LIN {X 0,Y 115.903,Z 1227.166,A -85,B 0,C 180,E1 30525.083,E2 30525.083} C_VEL
LIN {X 0,Y 121.307,Z 1221.826,A -85,B 0,C 180,E1 30544.058,E2 30544.058} C_VEL
LIN {X 0,Y 149.236,Z 1207.445,A -85,B 0,C 180,E1 30568.46,E2 30568.46} C_VEL
LIN {X 0,Y 160.737,Z 1202.235,A -85,B 0,C 180,E1 30574.059,E2 30574.059} C_VEL
LIN {X 0,Y 129.923,Z 1200.348,A -85,B 0,C 180,E1 30593.319,E2 30593.319} C_VEL
LIN {X 0,Y 116.524,Z 1195.812,A -85,B 0,C 180,E1 30615.028,E2 30615.028} C_VEL
LIN {X 0,Y 115.852,Z 1188.978,A -85,B 0,C 180,E1 30635.424,E2 30635.424} C_VEL
LIN {X 0,Y 122.473,Z 1180.721,A -85,B 0,C 180,E1 30651.947,E2 30651.947} C_VEL
LIN {X 0,Y 138.737,Z 1166.544,A -85,B 0,C 180,E1 30669.914,E2 30669.914} C_VEL
LIN {X 0,Y 165.96,Z 1145.332,A -85,B 0,C 180,E1 30684.797,E2 30684.797} C_VEL
LIN {X 0,Y 197.116,Z 1119.047,A -85,B 0,C 180,E1 30694.805,E2 30694.805} C_VEL
LIN {X 0,Y 228.825,Z 1088.466,A -85,B 0,C 180,E1 30701.734,E2 30701.734} C_VEL
LIN {X 0,Y 247.509,Z 1067.925,A -85,B 0,C 180,E1 30704.862,E2 30704.862} C_VEL
LIN {X 0,Y 250.073,Z 1055.769,A -85,B 0,C 180,E1 30711.272,E2 30711.272} C_VEL
LIN {X 0,Y 251.256,Z 1045.915,A -85,B 0,C 180,E1 30717.768,E2 30717.768} C_VEL
LIN {X 0,Y 251.874,Z 1037.298,A -85,B 0,C 180,E1 30725.345,E2 30725.345} C_VEL
LIN {X 0,Y 252.29,Z 1032.887,A -85,B 0,C 180,E1 30731.229,E2 30731.229} C_VEL
LIN {X 0,Y 252.785,Z 1030.009,A -85,B 0,C 180,E1 30738.891,E2 30738.891} C_VEL
LIN {X 0,Y 253.685,Z 1029.517,A -85,B 0,C 180,E1 30744.152,E2 30744.152} C_VEL
LIN {X 0,Y 252.999,Z 1031.73,A -85,B 0,C 180,E1 30747.067,E2 30747.067} C_VEL
LIN {X 0,Y 251.361,Z 1037.125,A -85,B 0,C 180,E1 30751.921,E2 30751.921} C_VEL
LIN {X 0,Y 254.488,Z 1040.821,A -85,B 0,C 180,E1 30759.132,E2 30759.132} C_VEL
LIN {X 0,Y 258.114,Z 1049.252,A -85,B 0,C 180,E1 30767.246,E2 30767.246} C_VEL
LIN {X 0,Y 260.709,Z 1059.906,A -85,B 0,C 180,E1 30773.967,E2 30773.967} C_VEL
LIN {X 0,Y 263.22,Z 1075.308,A -85,B 0,C 180,E1 30781.406,E2 30781.406} C_VEL
LIN {X 0,Y 263.374,Z 1076.931,A -85,B 0,C 180,E1 30782.108,E2 30782.108} C_VEL
LIN {X 0,Y 229.491,Z 1117.049,A -85,B 0,C 180,E1 30786.492,E2 30786.492} C_VEL
LIN {X 0,Y 196.364,Z 1149.598,A -85,B 0,C 180,E1 30792.406,E2 30792.406} C_VEL
LIN {X 0,Y 164.117,Z 1177.145,A -85,B 0,C 180,E1 30801.157,E2 30801.157} C_VEL
LIN {X 0,Y 136.729,Z 1198.115,A -85,B 0,C 180,E1 30813.545,E2 30813.545} C_VEL
LIN {X 0,Y 117.332,Z 1213.51,A -85,B 0,C 180,E1 30830.599,E2 30830.599} C_VEL
LIN {X 0,Y 109.107,Z 1222.749,A -85,B 0,C 180,E1 30849.709,E2 30849.709} C_VEL
LIN {X 0,Y 108.282,Z 1226.006,A -85,B 0,C 180,E1 30861.945,E2 30861.945} C_VEL
LIN {X 0,Y 109.205,Z 1227.073,A -85,B 0,C 180,E1 30869.968,E2 30869.968} C_VEL
LIN {X 0,Y 108.146,Z 1225.726,A -85,B 0,C 180,E1 30886.193,E2 30886.193} C_VEL
LIN {X 0,Y 115.945,Z 1219.699,A -85,B 0,C 180,E1 30908.559,E2 30908.559} C_VEL
LIN {X 0,Y 148.879,Z 1205.076,A -85,B 0,C 180,E1 30933.089,E2 30933.089} C_VEL
LIN {X 0,Y 150.497,Z 1204.236,A -85,B 0,C 180,E1 30934.137,E2 30934.137} C_VEL
LIN {X 0,Y 121.73,Z 1201.678,A -85,B 0,C 180,E1 30952.998,E2 30952.998} C_VEL
LIN {X 0,Y 108.299,Z 1196.353,A -85,B 0,C 180,E1 30976.2,E2 30976.2} C_VEL
LIN {X 0,Y 108.593,Z 1188.984,A -85,B 0,C 180,E1 30997.991,E2 30997.991} C_VEL
LIN {X 0,Y 116.696,Z 1180.045,A -85,B 0,C 180,E1 31015.734,E2 31015.734} C_VEL
LIN {X 0,Y 137.512,Z 1163.474,A -85,B 0,C 180,E1 31035.364,E2 31035.364} C_VEL
LIN {X 0,Y 166.233,Z 1141.644,A -85,B 0,C 180,E1 31048.906,E2 31048.906} C_VEL
LIN {X 0,Y 198.392,Z 1114.848,A -85,B 0,C 180,E1 31058.079,E2 31058.079} C_VEL
LIN {X 0,Y 232.591,Z 1081.271,A -85,B 0,C 180,E1 31064.742,E2 31064.742} C_VEL
LIN {X 0,Y 242.121,Z 1070.542,A -85,B 0,C 180,E1 31066.39,E2 31066.39} C_VEL
LIN {X 0,Y 244.698,Z 1059.241,A -85,B 0,C 180,E1 31072.716,E2 31072.716} C_VEL
LIN {X 0,Y 245.996,Z 1049.786,A -85,B 0,C 180,E1 31079.449,E2 31079.449} C_VEL
LIN {X 0,Y 247.016,Z 1041.487,A -85,B 0,C 180,E1 31087.732,E2 31087.732} C_VEL
LIN {X 0,Y 247.351,Z 1038.331,A -85,B 0,C 180,E1 31092.86,E2 31092.86} C_VEL
LIN {X 0,Y 248.6,Z 1035.925,A -85,B 0,C 180,E1 31102.224,E2 31102.224} C_VEL
LIN {X 0,Y 251.159,Z 1036.873,A -85,B 0,C 180,E1 31111.232,E2 31111.232} C_VEL
LIN {X 0,Y 251.361,Z 1037.125,A -85,B 0,C 180,E1 31111.921,E2 31111.921} C_VEL
LIN {X 0,Y 251.021,Z 1040.302,A -85,B 0,C 180,E1 31114.822,E2 31114.822} C_VEL
LIN {X 0,Y 249.783,Z 1047.533,A -85,B 0,C 180,E1 31119.608,E2 31119.608} C_VEL
LIN {X 0,Y 253.284,Z 1056.269,A -85,B 0,C 180,E1 31127.95,E2 31127.95} C_VEL
LIN {X 0,Y 255.662,Z 1067.949,A -85,B 0,C 180,E1 31135.014,E2 31135.014} C_VEL
LIN {X 0,Y 256.974,Z 1080.351,A -85,B 0,C 180,E1 31140.941,E2 31140.941} C_VEL
LIN {X 0,Y 223.473,Z 1118.609,A -85,B 0,C 180,E1 31145.07,E2 31145.07} C_VEL
LIN {X 0,Y 186.796,Z 1153.281,A -85,B 0,C 180,E1 31151.557,E2 31151.557} C_VEL
LIN {X 0,Y 154.639,Z 1179.212,A -85,B 0,C 180,E1 31160.504,E2 31160.504} C_VEL
LIN {X 0,Y 127.088,Z 1199.404,A -85,B 0,C 180,E1 31173.616,E2 31173.616} C_VEL
LIN {X 0,Y 108.285,Z 1213.812,A -85,B 0,C 180,E1 31191.784,E2 31191.784} C_VEL
LIN {X 0,Y 100.902,Z 1222.307,A -85,B 0,C 180,E1 31212.535,E2 31212.535} C_VEL
LIN {X 0,Y 101.407,Z 1225.453,A -85,B 0,C 180,E1 31229.965,E2 31229.965} C_VEL
LIN {X 0,Y 100.398,Z 1224.298,A -85,B 0,C 180,E1 31247.481,E2 31247.481} C_VEL
LIN {X 0,Y 107.237,Z 1219.449,A -85,B 0,C 180,E1 31267.89,E2 31267.89} C_VEL
LIN {X 0,Y 136.554,Z 1207.341,A -85,B 0,C 180,E1 31292.225,E2 31292.225} C_VEL
LIN {X 0,Y 139.784,Z 1205.877,A -85,B 0,C 180,E1 31294.379,E2 31294.379} C_VEL
LIN {X 0,Y 107.624,Z 1201.286,A -85,B 0,C 180,E1 31319.997,E2 31319.997} C_VEL
LIN {X 0,Y 99.274,Z 1194.993,A -85,B 0,C 180,E1 31344.128,E2 31344.128} C_VEL
LIN {X 0,Y 103.71,Z 1186.418,A -85,B 0,C 180,E1 31366.753,E2 31366.753} C_VEL
LIN {X 0,Y 116.196,Z 1175.396,A -85,B 0,C 180,E1 31385.536,E2 31385.536} C_VEL
LIN {X 0,Y 141.482,Z 1157.033,A -85,B 0,C 180,E1 31402.985,E2 31402.985} C_VEL
LIN {X 0,Y 172.324,Z 1133.681,A -85,B 0,C 180,E1 31414.551,E2 31414.551} C_VEL
LIN {X 0,Y 205.729,Z 1105.109,A -85,B 0,C 180,E1 31422.412,E2 31422.412} C_VEL
LIN {X 0,Y 236.572,Z 1073.596,A -85,B 0,C 180,E1 31427.744,E2 31427.744} C_VEL
LIN {X 0,Y 239.332,Z 1062.684,A -85,B 0,C 180,E1 31434.245,E2 31434.245} C_VEL
LIN {X 0,Y 240.84,Z 1053.518,A -85,B 0,C 180,E1 31441.491,E2 31441.491} C_VEL
LIN {X 0,Y 241.954,Z 1046.947,A -85,B 0,C 180,E1 31448.665,E2 31448.665} C_VEL
LIN {X 0,Y 242.687,Z 1043.093,A -85,B 0,C 180,E1 31456.777,E2 31456.777} C_VEL
LIN {X 0,Y 244.616,Z 1042.241,A -85,B 0,C 180,E1 31466.227,E2 31466.227} C_VEL
LIN {X 0,Y 247.713,Z 1044.501,A -85,B 0,C 180,E1 31474.725,E2 31474.725} C_VEL
LIN {X 0,Y 249.783,Z 1047.533,A -85,B 0,C 180,E1 31479.608,E2 31479.608} C_VEL
LIN {X 0,Y 249.353,Z 1051.979,A -85,B 0,C 180,E1 31482.44,E2 31482.44} C_VEL
LIN {X 0,Y 247.711,Z 1061.226,A -85,B 0,C 180,E1 31487.083,E2 31487.083} C_VEL
LIN {X 0,Y 249.801,Z 1071.906,A -85,B 0,C 180,E1 31493.925,E2 31493.925} C_VEL
LIN {X 0,Y 251.125,Z 1082.686,A -85,B 0,C 180,E1 31499.497,E2 31499.497} C_VEL
LIN {X 0,Y 220.201,Z 1117.408,A -85,B 0,C 180,E1 31503.214,E2 31503.214} C_VEL
LIN {X 0,Y 182.355,Z 1152.44,A -85,B 0,C 180,E1 31509.541,E2 31509.541} C_VEL
LIN {X 0,Y 148.605,Z 1178.767,A -85,B 0,C 180,E1 31518.583,E2 31518.583} C_VEL
LIN {X 0,Y 120.171,Z 1198.668,A -85,B 0,C 180,E1 31531.868,E2 31531.868} C_VEL
LIN {X 0,Y 101.316,Z 1212.21,A -85,B 0,C 180,E1 31549.776,E2 31549.776} C_VEL
LIN {X 0,Y 93.27,Z 1220.523,A -85,B 0,C 180,E1 31571.054,E2 31571.054} C_VEL
LIN {X 0,Y 93.589,Z 1223.855,A -85,B 0,C 180,E1 31589.962,E2 31589.962} C_VEL
LIN {X 0,Y 92.711,Z 1222.762,A -85,B 0,C 180,E1 31608.984,E2 31608.984} C_VEL
LIN {X 0,Y 104.857,Z 1216.407,A -85,B 0,C 180,E1 31636.049,E2 31636.049} C_VEL
LIN {X 0,Y 129.649,Z 1207.413,A -85,B 0,C 180,E1 31654.348,E2 31654.348} C_VEL
LIN {X 0,Y 99.287,Z 1202.08,A -85,B 0,C 180,E1 31679.997,E2 31679.997} C_VEL
LIN {X 0,Y 91.371,Z 1195.363,A -85,B 0,C 180,E1 31705.839,E2 31705.839} C_VEL
LIN {X 0,Y 96.333,Z 1187.072,A -85,B 0,C 180,E1 31728.41,E2 31728.41} C_VEL
LIN {X 0,Y 110.812,Z 1175.137,A -85,B 0,C 180,E1 31748.955,E2 31748.955} C_VEL
LIN {X 0,Y 137.994,Z 1156.444,A -85,B 0,C 180,E1 31766.214,E2 31766.214} C_VEL
LIN {X 0,Y 171.971,Z 1131.211,A -85,B 0,C 180,E1 31777.815,E2 31777.815} C_VEL
LIN {X 0,Y 205.821,Z 1102.143,A -85,B 0,C 180,E1 31785.048,E2 31785.048} C_VEL
LIN {X 0,Y 231.083,Z 1076.83,A -85,B 0,C 180,E1 31789.1,E2 31789.1} C_VEL
LIN {X 0,Y 234.064,Z 1066.08,A -85,B 0,C 180,E1 31795.989,E2 31795.989} C_VEL
LIN {X 0,Y 235.794,Z 1057.293,A -85,B 0,C 180,E1 31803.589,E2 31803.589} C_VEL
LIN {X 0,Y 236.788,Z 1052.096,A -85,B 0,C 180,E1 31810.029,E2 31810.029} C_VEL
LIN {X 0,Y 237.495,Z 1049.645,A -85,B 0,C 180,E1 31815.588,E2 31815.588} C_VEL
LIN {X 0,Y 239.297,Z 1048.305,A -85,B 0,C 180,E1 31825.2,E2 31825.2} C_VEL
LIN {X 0,Y 242.39,Z 1050.363,A -85,B 0,C 180,E1 31834.13,E2 31834.13} C_VEL
LIN {X 0,Y 244.886,Z 1053.918,A -85,B 0,C 180,E1 31840.029,E2 31840.029} C_VEL
LIN {X 0,Y 247.711,Z 1061.226,A -85,B 0,C 180,E1 31847.083,E2 31847.083} C_VEL
LIN {X 0,Y 246.931,Z 1067.057,A -85,B 0,C 180,E1 31849.812,E2 31849.812} C_VEL
LIN {X 0,Y 244.195,Z 1078.298,A -85,B 0,C 180,E1 31854.237,E2 31854.237} C_VEL
LIN {X 0,Y 244.491,Z 1086.498,A -85,B 0,C 180,E1 31858.263,E2 31858.263} C_VEL
LIN {X 0,Y 209.883,Z 1123.195,A -85,B 0,C 180,E1 31862.262,E2 31862.262} C_VEL
LIN {X 0,Y 174.487,Z 1154.462,A -85,B 0,C 180,E1 31868.179,E2 31868.179} C_VEL
LIN {X 0,Y 139.774,Z 1180.356,A -85,B 0,C 180,E1 31877.532,E2 31877.532} C_VEL
LIN {X 0,Y 110.922,Z 1199.471,A -85,B 0,C 180,E1 31891.574,E2 31891.574} C_VEL
LIN {X 0,Y 90.556,Z 1213.571,A -85,B 0,C 180,E1 31914.224,E2 31914.224} C_VEL
LIN {X 0,Y 84.916,Z 1220.325,A -85,B 0,C 180,E1 31936.947,E2 31936.947} C_VEL
LIN {X 0,Y 85.769,Z 1222.218,A -85,B 0,C 180,E1 31949.959,E2 31949.959} C_VEL
LIN {X 0,Y 85.128,Z 1221.178,A -85,B 0,C 180,E1 31970.749,E2 31970.749} C_VEL
LIN {X 0,Y 99.219,Z 1215.064,A -85,B 0,C 180,E1 31999.539,E2 31999.539} C_VEL
LIN {X 0,Y 118.108,Z 1208.948,A -85,B 0,C 180,E1 32013.513,E2 32013.513} C_VEL
LIN {X 0,Y 118.736,Z 1208.442,A -85,B 0,C 180,E1 32014.648,E2 32014.648} C_VEL
LIN {X 0,Y 90.605,Z 1202.768,A -85,B 0,C 180,E1 32040.532,E2 32040.532} C_VEL
LIN {X 0,Y 83.576,Z 1195.469,A -85,B 0,C 180,E1 32068.735,E2 32068.735} C_VEL
LIN {X 0,Y 90.422,Z 1186.476,A -85,B 0,C 180,E1 32093.096,E2 32093.096} C_VEL
LIN {X 0,Y 109.279,Z 1172.666,A -85,B 0,C 180,E1 32115.427,E2 32115.427} C_VEL
LIN {X 0,Y 138.694,Z 1153.021,A -85,B 0,C 180,E1 32131.101,E2 32131.101} C_VEL
LIN {X 0,Y 171.661,Z 1128.922,A -85,B 0,C 180,E1 32140.994,E2 32140.994} C_VEL
LIN {X 0,Y 209.084,Z 1096.491,A -85,B 0,C 180,E1 32148.146,E2 32148.146} C_VEL
LIN {X 0,Y 225.667,Z 1079.947,A -85,B 0,C 180,E1 32150.598,E2 32150.598} C_VEL
LIN {X 0,Y 228.771,Z 1069.776,A -85,B 0,C 180,E1 32157.556,E2 32157.556} C_VEL
LIN {X 0,Y 230.922,Z 1060.913,A -85,B 0,C 180,E1 32166.099,E2 32166.099} C_VEL
LIN {X 0,Y 232.082,Z 1056.025,A -85,B 0,C 180,E1 32174.263,E2 32174.263} C_VEL
LIN {X 0,Y 233.247,Z 1054.561,A -85,B 0,C 180,E1 32181.047,E2 32181.047} C_VEL
LIN {X 0,Y 235.455,Z 1054.955,A -85,B 0,C 180,E1 32189.112,E2 32189.112} C_VEL
LIN {X 0,Y 238.834,Z 1058.342,A -85,B 0,C 180,E1 32197.693,E2 32197.693} C_VEL
LIN {X 0,Y 241.94,Z 1065.38,A -85,B 0,C 180,E1 32205.535,E2 32205.535} C_VEL
LIN {X 0,Y 243.76,Z 1074.732,A -85,B 0,C 180,E1 32212.154,E2 32212.154} C_VEL
LIN {X 0,Y 244.195,Z 1078.298,A -85,B 0,C 180,E1 32214.237,E2 32214.237} C_VEL
LIN {X 0,Y 242.463,Z 1083.265,A -85,B 0,C 180,E1 32215.784,E2 32215.784} C_VEL
LIN {X 0,Y 235.136,Z 1093.065,A -85,B 0,C 180,E1 32217.169,E2 32217.169} C_VEL
LIN {X 0,Y 225.579,Z 1103.372,A -85,B 0,C 180,E1 32218.121,E2 32218.121} C_VEL
LIN {X 0,Y 187.741,Z 1139.371,A -85,B 0,C 180,E1 32222.924,E2 32222.924} C_VEL
LIN {X 0,Y 150.886,Z 1168.156,A -85,B 0,C 180,E1 32230.295,E2 32230.295} C_VEL
LIN {X 0,Y 117.953,Z 1190.195,A -85,B 0,C 180,E1 32241.676,E2 32241.676} C_VEL
LIN {X 0,Y 89.807,Z 1207.468,A -85,B 0,C 180,E1 32262.303,E2 32262.303} C_VEL
LIN {X 0,Y 78.256,Z 1216.707,A -85,B 0,C 180,E1 32287.234,E2 32287.234} C_VEL
LIN {X 0,Y 77.955,Z 1220.615,A -85,B 0,C 180,E1 32309.955,E2 32309.955} C_VEL
LIN {X 0,Y 77.617,Z 1219.589,A -85,B 0,C 180,E1 32332.865,E2 32332.865} C_VEL
LIN {X 0,Y 93.973,Z 1213.764,A -85,B 0,C 180,E1 32363.449,E2 32363.449} C_VEL
LIN {X 0,Y 107.273,Z 1209.979,A -85,B 0,C 180,E1 32373.353,E2 32373.353} C_VEL
LIN {X 0,Y 107.65,Z 1209.322,A -85,B 0,C 180,E1 32375.094,E2 32375.094} C_VEL
LIN {X 0,Y 82.522,Z 1203.513,A -85,B 0,C 180,E1 32399.996,E2 32399.996} C_VEL
LIN {X 0,Y 75.939,Z 1195.293,A -85,B 0,C 180,E1 32432.258,E2 32432.258} C_VEL
LIN {X 0,Y 82.212,Z 1187.978,A -85,B 0,C 180,E1 32453.266,E2 32453.266} C_VEL
LIN {X 0,Y 101.88,Z 1174.273,A -85,B 0,C 180,E1 32477.108,E2 32477.108} C_VEL
LIN {X 0,Y 134.837,Z 1153.139,A -85,B 0,C 180,E1 32494.061,E2 32494.061} C_VEL
LIN {X 0,Y 170.155,Z 1127.672,A -85,B 0,C 180,E1 32503.804,E2 32503.804} C_VEL
LIN {X 0,Y 206.882,Z 1096.207,A -85,B 0,C 180,E1 32510.281,E2 32510.281} C_VEL
LIN {X 0,Y 220.284,Z 1083.018,A -85,B 0,C 180,E1 32512.182,E2 32512.182} C_VEL
LIN {X 0,Y 223.508,Z 1073.292,A -85,B 0,C 180,E1 32519.404,E2 32519.404} C_VEL
LIN {X 0,Y 225.548,Z 1065.936,A -85,B 0,C 180,E1 32527.101,E2 32527.101} C_VEL
LIN {X 0,Y 226.561,Z 1062.682,A -85,B 0,C 180,E1 32532.812,E2 32532.812} C_VEL
LIN {X 0,Y 227.429,Z 1060.907,A -85,B 0,C 180,E1 32538.367,E2 32538.367} C_VEL
LIN {X 0,Y 229.966,Z 1060.819,A -85,B 0,C 180,E1 32548.29,E2 32548.29} C_VEL
LIN {X 0,Y 233.412,Z 1064.015,A -85,B 0,C 180,E1 32557.146,E2 32557.146} C_VEL
LIN {X 0,Y 235.899,Z 1069.552,A -85,B 0,C 180,E1 32563.963,E2 32563.963} C_VEL
LIN {X 0,Y 237.722,Z 1076.998,A -85,B 0,C 180,E1 32569.935,E2 32569.935} C_VEL
LIN {X 0,Y 238.922,Z 1088.606,A -85,B 0,C 180,E1 32576.717,E2 32576.717} C_VEL
LIN {X 0,Y 225.579,Z 1103.372,A -85,B 0,C 180,E1 32578.121,E2 32578.121} C_VEL
LIN {X 0,Y 212.287,Z 1114.899,A -85,B 0,C 180,E1 32578.46,E2 32578.46} C_VEL
LIN {X 0,Y 198.702,Z 1125.77,A -85,B 0,C 180,E1 32578.863,E2 32578.863} C_VEL
LIN {X 0,Y 159.946,Z 1157.516,A -85,B 0,C 180,E1 32584.887,E2 32584.887} C_VEL
LIN {X 0,Y 124.697,Z 1181.57,A -85,B 0,C 180,E1 32594.091,E2 32594.091} C_VEL
LIN {X 0,Y 92.777,Z 1200.371,A -85,B 0,C 180,E1 32610.453,E2 32610.453} C_VEL
LIN {X 0,Y 74.097,Z 1212.072,A -85,B 0,C 180,E1 32634.662,E2 32634.662} C_VEL
LIN {X 0,Y 69.433,Z 1217.316,A -85,B 0,C 180,E1 32657.378,E2 32657.378} C_VEL
LIN {X 0,Y 70.124,Z 1218.977,A -85,B 0,C 180,E1 32669.95,E2 32669.95} C_VEL
LIN {X 0,Y 70.212,Z 1218.018,A -85,B 0,C 180,E1 32695.439,E2 32695.439} C_VEL
LIN {X 0,Y 93.075,Z 1211.415,A -85,B 0,C 180,E1 32730.851,E2 32730.851} C_VEL
LIN {X 0,Y 97.648,Z 1209.934,A -85,B 0,C 180,E1 32734.812,E2 32734.812} C_VEL
LIN {X 0,Y 71.413,Z 1202.635,A -85,B 0,C 180,E1 32766.068,E2 32766.068} C_VEL
LIN {X 0,Y 69.467,Z 1193.839,A -85,B 0,C 180,E1 32800.727,E2 32800.727} C_VEL
LIN {X 0,Y 82.179,Z 1183.556,A -85,B 0,C 180,E1 32826.817,E2 32826.817} C_VEL
LIN {X 0,Y 108.192,Z 1167.625,A -85,B 0,C 180,E1 32847.624,E2 32847.624} C_VEL
LIN {X 0,Y 144.99,Z 1144.018,A -85,B 0,C 180,E1 32861.233,E2 32861.233} C_VEL
LIN {X 0,Y 181.817,Z 1116.16,A -85,B 0,C 180,E1 32868.972,E2 32868.972} C_VEL
LIN {X 0,Y 214.456,Z 1086.665,A -85,B 0,C 180,E1 32873.664,E2 32873.664} C_VEL
LIN {X 0,Y 217.473,Z 1079.22,A -85,B 0,C 180,E1 32879.121,E2 32879.121} C_VEL
LIN {X 0,Y 219.944,Z 1071.907,A -85,B 0,C 180,E1 32886.803,E2 32886.803} C_VEL
LIN {X 0,Y 221.145,Z 1068.344,A -85,B 0,C 180,E1 32893.122,E2 32893.122} C_VEL
LIN {X 0,Y 222.22,Z 1066.806,A -85,B 0,C 180,E1 32898.439,E2 32898.439} C_VEL
LIN {X 0,Y 224.377,Z 1066.687,A -85,B 0,C 180,E1 32907.404,E2 32907.404} C_VEL
LIN {X 0,Y 227.864,Z 1069.547,A -85,B 0,C 180,E1 32916.557,E2 32916.557} C_VEL
LIN {X 0,Y 230.348,Z 1075.001,A -85,B 0,C 180,E1 32923.565,E2 32923.565} C_VEL
LIN {X 0,Y 232.09,Z 1082.623,A -85,B 0,C 180,E1 32929.785,E2 32929.785} C_VEL
LIN {X 0,Y 232.708,Z 1091.127,A -85,B 0,C 180,E1 32935.051,E2 32935.051} C_VEL
LIN {X 0,Y 226.294,Z 1098.652,A -85,B 0,C 180,E1 32935.885,E2 32935.885} C_VEL
LIN {X 0,Y 198.702,Z 1125.77,A -85,B 0,C 180,E1 32938.863,E2 32938.863} C_VEL
LIN {X 0,Y 184.688,Z 1136.141,A -85,B 0,C 180,E1 32939.397,E2 32939.397} C_VEL
LIN {X 0,Y 170.262,Z 1145.957,A -85,B 0,C 180,E1 32940.057,E2 32940.057} C_VEL
LIN {X 0,Y 133.367,Z 1172.138,A -85,B 0,C 180,E1 32947.327,E2 32947.327} C_VEL
LIN {X 0,Y 97.017,Z 1193.556,A -85,B 0,C 180,E1 32960.749,E2 32960.749} C_VEL
LIN {X 0,Y 71.964,Z 1207.28,A -85,B 0,C 180,E1 32982.628,E2 32982.628} C_VEL
LIN {X 0,Y 62.318,Z 1214.25,A -85,B 0,C 180,E1 33008.611,E2 33008.611} C_VEL
LIN {X 0,Y 62.286,Z 1217.241,A -85,B 0,C 180,E1 33029.943,E2 33029.943} C_VEL
LIN {X 0,Y 62.981,Z 1216.434,A -85,B 0,C 180,E1 33058.611,E2 33058.611} C_VEL
LIN {X 0,Y 85.05,Z 1210.99,A -85,B 0,C 180,E1 33092.573,E2 33092.573} C_VEL
LIN {X 0,Y 86.971,Z 1210.32,A -85,B 0,C 180,E1 33094.867,E2 33094.867} C_VEL
LIN {X 0,Y 63.358,Z 1203.125,A -85,B 0,C 180,E1 33125.639,E2 33125.639} C_VEL
LIN {X 0,Y 62.006,Z 1194.281,A -85,B 0,C 180,E1 33163.107,E2 33163.107} C_VEL
LIN {X 0,Y 75.048,Z 1184.579,A -85,B 0,C 180,E1 33189.297,E2 33189.297} C_VEL
LIN {X 0,Y 103.396,Z 1168.146,A -85,B 0,C 180,E1 33211.019,E2 33211.019} C_VEL
LIN {X 0,Y 139.95,Z 1145.455,A -85,B 0,C 180,E1 33223.675,E2 33223.675} C_VEL
LIN {X 0,Y 176.173,Z 1118.825,A -85,B 0,C 180,E1 33230.853,E2 33230.853} C_VEL
LIN {X 0,Y 208.619,Z 1090.236,A -85,B 0,C 180,E1 33235.293,E2 33235.293} C_VEL
LIN {X 0,Y 210.273,Z 1087.701,A -85,B 0,C 180,E1 33236.707,E2 33236.707} C_VEL
LIN {X 0,Y 213.099,Z 1080.328,A -85,B 0,C 180,E1 33243.61,E2 33243.61} C_VEL
LIN {X 0,Y 214.847,Z 1076.069,A -85,B 0,C 180,E1 33249.323,E2 33249.323} C_VEL
LIN {X 0,Y 216.09,Z 1073.307,A -85,B 0,C 180,E1 33255.636,E2 33255.636} C_VEL
LIN {X 0,Y 217.309,Z 1072.331,A -85,B 0,C 180,E1 33261.262,E2 33261.262} C_VEL
LIN {X 0,Y 220.47,Z 1073.36,A -85,B 0,C 180,E1 33271.333,E2 33271.333} C_VEL
LIN {X 0,Y 222.837,Z 1075.874,A -85,B 0,C 180,E1 33277.339,E2 33277.339} C_VEL
LIN {X 0,Y 225.171,Z 1081.574,A -85,B 0,C 180,E1 33284.432,E2 33284.432} C_VEL
LIN {X 0,Y 226.324,Z 1089.454,A -85,B 0,C 180,E1 33290.593,E2 33290.593} C_VEL
LIN {X 0,Y 226.612,Z 1094.256,A -85,B 0,C 180,E1 33293.599,E2 33293.599} C_VEL
LIN {X 0,Y 192.952,Z 1127.191,A -85,B 0,C 180,E1 33297.063,E2 33297.063} C_VEL
LIN {X 0,Y 170.262,Z 1145.957,A -85,B 0,C 180,E1 33300.057,E2 33300.057} C_VEL
LIN {X 0,Y 155.555,Z 1155.214,A -85,B 0,C 180,E1 33300.903,E2 33300.903} C_VEL
LIN {X 0,Y 140.47,Z 1163.805,A -85,B 0,C 180,E1 33301.983,E2 33301.983} C_VEL
LIN {X 0,Y 103.19,Z 1186.283,A -85,B 0,C 180,E1 33312.204,E2 33312.204} C_VEL
LIN {X 0,Y 71.348,Z 1202.56,A -85,B 0,C 180,E1 33332.004,E2 33332.004} C_VEL
LIN {X 0,Y 56.729,Z 1210.88,A -85,B 0,C 180,E1 33357.737,E2 33357.737} C_VEL
LIN {X 0,Y 54.477,Z 1215.425,A -85,B 0,C 180,E1 33389.935,E2 33389.935} C_VEL
LIN {X 0,Y 55.956,Z 1214.798,A -85,B 0,C 180,E1 33422.614,E2 33422.614} C_VEL
LIN {X 0,Y 76.462,Z 1210.365,A -85,B 0,C 180,E1 33454.737,E2 33454.737} C_VEL
LIN {X 0,Y 53.408,Z 1201.994,A -85,B 0,C 180,E1 33492.642,E2 33492.642} C_VEL
LIN {X 0,Y 58.364,Z 1191.678,A -85,B 0,C 180,E1 33536.352,E2 33536.352} C_VEL
LIN {X 0,Y 76.492,Z 1180.816,A -85,B 0,C 180,E1 33560.968,E2 33560.968} C_VEL
LIN {X 0,Y 110.167,Z 1162.306,A -85,B 0,C 180,E1 33579.149,E2 33579.149} C_VEL
LIN {X 0,Y 150.078,Z 1136.774,A -85,B 0,C 180,E1 33589.463,E2 33589.463} C_VEL
LIN {X 0,Y 187.888,Z 1107.354,A -85,B 0,C 180,E1 33595.22,E2 33595.22} C_VEL
LIN {X 0,Y 203.641,Z 1093.176,A -85,B 0,C 180,E1 33597.082,E2 33597.082} C_VEL
LIN {X 0,Y 206.166,Z 1088.479,A -85,B 0,C 180,E1 33600.887,E2 33600.887} C_VEL
LIN {X 0,Y 208.503,Z 1082.984,A -85,B 0,C 180,E1 33607.144,E2 33607.144} C_VEL
LIN {X 0,Y 210.657,Z 1078.997,A -85,B 0,C 180,E1 33615.856,E2 33615.856} C_VEL
LIN {X 0,Y 212.832,Z 1078.121,A -85,B 0,C 180,E1 33625.394,E2 33625.394} C_VEL
LIN {X 0,Y 214.535,Z 1078.875,A -85,B 0,C 180,E1 33630.463,E2 33630.463} C_VEL
LIN {X 0,Y 217.078,Z 1081.224,A -85,B 0,C 180,E1 33636.824,E2 33636.824} C_VEL
LIN {X 0,Y 219.521,Z 1087.322,A -85,B 0,C 180,E1 33644.57,E2 33644.57} C_VEL
LIN {X 0,Y 220.502,Z 1095.889,A -85,B 0,C 180,E1 33651.132,E2 33651.132} C_VEL
LIN {X 0,Y 220.578,Z 1097.445,A -85,B 0,C 180,E1 33652.127,E2 33652.127} C_VEL
LIN {X 0,Y 181.886,Z 1133.106,A -85,B 0,C 180,E1 33655.756,E2 33655.756} C_VEL
LIN {X 0,Y 143.653,Z 1161.712,A -85,B 0,C 180,E1 33661.381,E2 33661.381} C_VEL
LIN {X 0,Y 140.47,Z 1163.805,A -85,B 0,C 180,E1 33661.983,E2 33661.983} C_VEL
LIN {X 0,Y 125.189,Z 1171.835,A -85,B 0,C 180,E1 33663.353,E2 33663.353} C_VEL
LIN {X 0,Y 109.661,Z 1179.142,A -85,B 0,C 180,E1 33665.199,E2 33665.199} C_VEL
LIN {X 0,Y 73.08,Z 1197.551,A -85,B 0,C 180,E1 33681.363,E2 33681.363} C_VEL
LIN {X 0,Y 50.1,Z 1208.815,A -85,B 0,C 180,E1 33712.811,E2 33712.811} C_VEL
LIN {X 0,Y 46.646,Z 1213.626,A -85,B 0,C 180,E1 33749.924,E2 33749.924} C_VEL
LIN {X 0,Y 49.29,Z 1213.016,A -85,B 0,C 180,E1 33787.725,E2 33787.725} C_VEL
LIN {X 0,Y 65.807,Z 1210.193,A -85,B 0,C 180,E1 33814.494,E2 33814.494} C_VEL
LIN {X 0,Y 44.441,Z 1200.99,A -85,B 0,C 180,E1 33859.869,E2 33859.869} C_VEL
LIN {X 0,Y 53.698,Z 1190.781,A -85,B 0,C 180,E1 33904.794,E2 33904.794} C_VEL
LIN {X 0,Y 80.328,Z 1176.683,A -85,B 0,C 180,E1 33931.679,E2 33931.679} C_VEL
LIN {X 0,Y 117.533,Z 1156.348,A -85,B 0,C 180,E1 33946.021,E2 33946.021} C_VEL
LIN {X 0,Y 156.856,Z 1130.353,A -85,B 0,C 180,E1 33953.808,E2 33953.808} C_VEL
LIN {X 0,Y 194.318,Z 1100.238,A -85,B 0,C 180,E1 33958.497,E2 33958.497} C_VEL
LIN {X 0,Y 198.906,Z 1095.985,A -85,B 0,C 180,E1 33958.98,E2 33958.98} C_VEL
LIN {X 0,Y 202.478,Z 1088.957,A -85,B 0,C 180,E1 33966.678,E2 33966.678} C_VEL
LIN {X 0,Y 203.987,Z 1085.828,A -85,B 0,C 180,E1 33972.209,E2 33972.209} C_VEL
LIN {X 0,Y 205.5,Z 1084.055,A -85,B 0,C 180,E1 33978.569,E2 33978.569} C_VEL
LIN {X 0,Y 206.985,Z 1083.799,A -85,B 0,C 180,E1 33984.27,E2 33984.27} C_VEL
LIN {X 0,Y 208.941,Z 1084.507,A -85,B 0,C 180,E1 33990.241,E2 33990.241} C_VEL
LIN {X 0,Y 212.264,Z 1088.301,A -85,B 0,C 180,E1 33999.152,E2 33999.152} C_VEL
LIN {X 0,Y 214.207,Z 1094.848,A -85,B 0,C 180,E1 34006.336,E2 34006.336} C_VEL
LIN {X 0,Y 214.415,Z 1100.125,A -85,B 0,C 180,E1 34010.344,E2 34010.344} C_VEL
LIN {X 0,Y 176.8,Z 1134.045,A -85,B 0,C 180,E1 34013.665,E2 34013.665} C_VEL
LIN {X 0,Y 136.777,Z 1162.87,A -85,B 0,C 180,E1 34019.127,E2 34019.127} C_VEL
LIN {X 0,Y 109.661,Z 1179.142,A -85,B 0,C 180,E1 34025.199,E2 34025.199} C_VEL
LIN {X 0,Y 98.082,Z 1184.346,A -85,B 0,C 180,E1 34027.192,E2 34027.192} C_VEL
LIN {X 0,Y 79.932,Z 1190.847,A -85,B 0,C 180,E1 34030.195,E2 34030.195} C_VEL
LIN {X 0,Y 78.151,Z 1191.611,A -85,B 0,C 180,E1 34030.933,E2 34030.933} C_VEL
LIN {X 0,Y 49.023,Z 1204.258,A -85,B 0,C 180,E1 34055.864,E2 34055.864} C_VEL
LIN {X 0,Y 38.267,Z 1210.931,A -85,B 0,C 180,E1 34098.515,E2 34098.515} C_VEL
LIN {X 0,Y 38.816,Z 1211.791,A -85,B 0,C 180,E1 34109.909,E2 34109.909} C_VEL
LIN {X 0,Y 43.971,Z 1211.145,A -85,B 0,C 180,E1 34156.576,E2 34156.576} C_VEL
LIN {X 0,Y 51.995,Z 1210.193,A -85,B 0,C 180,E1 34170.534,E2 34170.534} C_VEL
LIN {X 0,Y 54.251,Z 1209.534,A -85,B 0,C 180,E1 34174.96,E2 34174.96} C_VEL
LIN {X 0,Y 36.318,Z 1200.652,A -85,B 0,C 180,E1 34224.575,E2 34224.575} C_VEL
LIN {X 0,Y 48.454,Z 1190.633,A -85,B 0,C 180,E1 34271.906,E2 34271.906} C_VEL
LIN {X 0,Y 78.366,Z 1176.018,A -85,B 0,C 180,E1 34297.697,E2 34297.697} C_VEL
LIN {X 0,Y 118.199,Z 1154.63,A -85,B 0,C 180,E1 34310.423,E2 34310.423} C_VEL
LIN {X 0,Y 161.563,Z 1125.709,A -85,B 0,C 180,E1 34317.473,E2 34317.473} C_VEL
LIN {X 0,Y 193.766,Z 1099.281,A -85,B 0,C 180,E1 34320.935,E2 34320.935} C_VEL
LIN {X 0,Y 196.889,Z 1093.57,A -85,B 0,C 180,E1 34327.9,E2 34327.9} C_VEL
LIN {X 0,Y 199.343,Z 1089.914,A -85,B 0,C 180,E1 34336.988,E2 34336.988} C_VEL
LIN {X 0,Y 201.586,Z 1089.462,A -85,B 0,C 180,E1 34345.573,E2 34345.573} C_VEL
LIN {X 0,Y 204.469,Z 1091.163,A -85,B 0,C 180,E1 34353.682,E2 34353.682} C_VEL
LIN {X 0,Y 206.777,Z 1094.427,A -85,B 0,C 180,E1 34360.027,E2 34360.027} C_VEL
LIN {X 0,Y 208.341,Z 1101.512,A -85,B 0,C 180,E1 34367.435,E2 34367.435} C_VEL
LIN {X 0,Y 208.352,Z 1103.021,A -85,B 0,C 180,E1 34368.552,E2 34368.552} C_VEL
LIN {X 0,Y 171.744,Z 1135.049,A -85,B 0,C 180,E1 34371.471,E2 34371.471} C_VEL
LIN {X 0,Y 128.857,Z 1164.785,A -85,B 0,C 180,E1 34376.868,E2 34376.868} C_VEL
LIN {X 0,Y 91.189,Z 1185.448,A -85,B 0,C 180,E1 34385.784,E2 34385.784} C_VEL
LIN {X 0,Y 78.151,Z 1191.611,A -85,B 0,C 180,E1 34390.933,E2 34390.933} C_VEL
LIN {X 0,Y 62.517,Z 1196.714,A -85,B 0,C 180,E1 34395.952,E2 34395.952} C_VEL
LIN {X 0,Y 47.257,Z 1200.977,A -85,B 0,C 180,E1 34404.109,E2 34404.109} C_VEL
LIN {X 0,Y 31.854,Z 1207.668,A -85,B 0,C 180,E1 34441.556,E2 34441.556} C_VEL
LIN {X 0,Y 30.944,Z 1209.973,A -85,B 0,C 180,E1 34469.886,E2 34469.886} C_VEL
LIN {X 0,Y 40.115,Z 1209.212,A -85,B 0,C 180,E1 34527.869,E2 34527.869} C_VEL
LIN {X 0,Y 43.07,Z 1208.581,A -85,B 0,C 180,E1 34534.966,E2 34534.966} C_VEL
LIN {X 0,Y 29.683,Z 1198.406,A -85,B 0,C 180,E1 34604.389,E2 34604.389} C_VEL
LIN {X 0,Y 49.31,Z 1188.145,A -85,B 0,C 180,E1 34646.536,E2 34646.536} C_VEL
LIN {X 0,Y 86.946,Z 1170.537,A -85,B 0,C 180,E1 34667.278,E2 34667.278} C_VEL
LIN {X 0,Y 128.272,Z 1147.456,A -85,B 0,C 180,E1 34676.207,E2 34676.207} C_VEL
LIN {X 0,Y 170.722,Z 1117.495,A -85,B 0,C 180,E1 34681.326,E2 34681.326} C_VEL
LIN {X 0,Y 188.574,Z 1102.729,A -85,B 0,C 180,E1 34683.006,E2 34683.006} C_VEL
LIN {X 0,Y 191.282,Z 1098.22,A -85,B 0,C 180,E1 34689.219,E2 34689.219} C_VEL
LIN {X 0,Y 193.045,Z 1095.887,A -85,B 0,C 180,E1 34695.218,E2 34695.218} C_VEL
LIN {X 0,Y 194.759,Z 1094.876,A -85,B 0,C 180,E1 34701.638,E2 34701.638} C_VEL
LIN {X 0,Y 196.549,Z 1095.19,A -85,B 0,C 180,E1 34707.777,E2 34707.777} C_VEL
LIN {X 0,Y 199.343,Z 1097.31,A -85,B 0,C 180,E1 34715.495,E2 34715.495} C_VEL
LIN {X 0,Y 201.608,Z 1101.797,A -85,B 0,C 180,E1 34722.557,E2 34722.557} C_VEL
LIN {X 0,Y 201.808,Z 1106.536,A -85,B 0,C 180,E1 34726.826,E2 34726.826} C_VEL
LIN {X 0,Y 163.615,Z 1138.336,A -85,B 0,C 180,E1 34729.492,E2 34729.492} C_VEL
LIN {X 0,Y 123.291,Z 1165.289,A -85,B 0,C 180,E1 34734.006,E2 34734.006} C_VEL
LIN {X 0,Y 83.258,Z 1186.053,A -85,B 0,C 180,E1 34742.651,E2 34742.651} C_VEL
LIN {X 0,Y 47.257,Z 1200.977,A -85,B 0,C 180,E1 34764.109,E2 34764.109} C_VEL
LIN {X 0,Y 36.954,Z 1203.779,A -85,B 0,C 180,E1 34774.594,E2 34774.594} C_VEL
LIN {X 0,Y 23.087,Z 1206.757,A -85,B 0,C 180,E1 34808.585,E2 34808.585} C_VEL
LIN {X 0,Y 23.08,Z 1208.051,A -85,B 0,C 180,E1 34829.847,E2 34829.847} C_VEL
LIN {X 0,Y 32.126,Z 1207.813,A -85,B 0,C 180,E1 34891.932,E2 34891.932} C_VEL
LIN {X 0,Y 20.587,Z 1201.812,A -85,B 0,C 180,E1 34941.512,E2 34941.512} C_VEL
LIN {X 0,Y 35.324,Z 1192.47,A -85,B 0,C 180,E1 35004.453,E2 35004.453} C_VEL
LIN {X 0,Y 71.842,Z 1176.908,A -85,B 0,C 180,E1 35028.645,E2 35028.645} C_VEL
LIN {X 0,Y 114.13,Z 1155.069,A -85,B 0,C 180,E1 35037.968,E2 35037.968} C_VEL
LIN {X 0,Y 157.482,Z 1126.755,A -85,B 0,C 180,E1 35042.938,E2 35042.938} C_VEL
LIN {X 0,Y 182.532,Z 1106.881,A -85,B 0,C 180,E1 35044.911,E2 35044.911} C_VEL
LIN {X 0,Y 184.481,Z 1104.63,A -85,B 0,C 180,E1 35047.384,E2 35047.384} C_VEL
LIN {X 0,Y 186.401,Z 1101.85,A -85,B 0,C 180,E1 35053.154,E2 35053.154} C_VEL
LIN {X 0,Y 189.167,Z 1100.274,A -85,B 0,C 180,E1 35063.046,E2 35063.046} C_VEL
LIN {X 0,Y 192.174,Z 1101.523,A -85,B 0,C 180,E1 35071.854,E2 35071.854} C_VEL
LIN {X 0,Y 194.722,Z 1104.29,A -85,B 0,C 180,E1 35078.673,E2 35078.673} C_VEL
LIN {X 0,Y 195.983,Z 1108.991,A -85,B 0,C 180,E1 35084.636,E2 35084.636} C_VEL
LIN {X 0,Y 160.17,Z 1138.291,A -85,B 0,C 180,E1 35086.927,E2 35086.927} C_VEL
LIN {X 0,Y 119.079,Z 1165.055,A -85,B 0,C 180,E1 35090.755,E2 35090.755} C_VEL
LIN {X 0,Y 79.448,Z 1184.906,A -85,B 0,C 180,E1 35097.847,E2 35097.847} C_VEL
LIN {X 0,Y 41.932,Z 1199.475,A -85,B 0,C 180,E1 35116.859,E2 35116.859} C_VEL
LIN {X 0,Y 23.087,Z 1206.757,A -85,B 0,C 180,E1 35168.585,E2 35168.585} C_VEL
LIN {X 0,Y 19.574,Z 1207.148,A -85,B 0,C 180,E1 35189.522,E2 35189.522} C_VEL
LIN {X 0,Y 17.634,Z 1206.172,A -85,B 0,C 180,E1 35238.159,E2 35238.159} C_VEL
LIN {X 0,Y 20.242,Z 1205.815,A -85,B 0,C 180,E1 35253.671,E2 35253.671} C_VEL
LIN {X 0,Y 26.094,Z 1194.703,A -85,B 0,C 180,E1 35370.136,E2 35370.136} C_VEL
LIN {X 0,Y 58.75,Z 1181.938,A -85,B 0,C 180,E1 35391.708,E2 35391.708} C_VEL
LIN {X 0,Y 102.427,Z 1161.065,A -85,B 0,C 180,E1 35400.64,E2 35400.64} C_VEL
LIN {X 0,Y 145.001,Z 1134.904,A -85,B 0,C 180,E1 35404.972,E2 35404.972} C_VEL
LIN {X 0,Y 178.059,Z 1109.891,A -85,B 0,C 180,E1 35407.235,E2 35407.235} C_VEL
LIN {X 0,Y 180.048,Z 1107.445,A -85,B 0,C 180,E1 35412.201,E2 35412.201} C_VEL
LIN {X 0,Y 181.842,Z 1105.905,A -85,B 0,C 180,E1 35418.435,E2 35418.435} C_VEL
LIN {X 0,Y 183.879,Z 1105.644,A -85,B 0,C 180,E1 35425.295,E2 35425.295} C_VEL
LIN {X 0,Y 186.543,Z 1107.117,A -85,B 0,C 180,E1 35433.044,E2 35433.044} C_VEL
LIN {X 0,Y 189.324,Z 1111.222,A -85,B 0,C 180,E1 35441.385,E2 35441.385} C_VEL
LIN {X 0,Y 189.514,Z 1112.262,A -85,B 0,C 180,E1 35442.62,E2 35442.62} C_VEL
LIN {X 0,Y 149.91,Z 1143.204,A -85,B 0,C 180,E1 35444.634,E2 35444.634} C_VEL
LIN {X 0,Y 106.192,Z 1169.567,A -85,B 0,C 180,E1 35448.196,E2 35448.196} C_VEL
LIN {X 0,Y 65.986,Z 1188.034,A -85,B 0,C 180,E1 35454.916,E2 35454.916} C_VEL
LIN {X 0,Y 31.183,Z 1199.964,A -85,B 0,C 180,E1 35473.8,E2 35473.8} C_VEL
LIN {X 0,Y 15.161,Z 1205.865,A -85,B 0,C 180,E1 35545.587,E2 35545.587} C_VEL
LIN {X 0,Y 17.634,Z 1206.172,A -85,B 0,C 180,E1 35598.159,E2 35598.159} C_VEL
LIN {X 0,Y 15.746,Z 1205.265,A -85,B 0,C 180,E1 35611.06,E2 35611.06} C_VEL
LIN {X 0,Y 7.96,Z 1200.101,A -85,B 0,C 180,E1 35720.575,E2 35720.575} C_VEL
LIN {X 0,Y 37.281,Z 1190,A -85,B 0,C 180,E1 35754.015,E2 35754.015} C_VEL
LIN {X 0,Y 82.909,Z 1170.788,A -85,B 0,C 180,E1 35763.196,E2 35763.196} C_VEL
LIN {X 0,Y 125.825,Z 1147.054,A -85,B 0,C 180,E1 35766.938,E2 35766.938} C_VEL
LIN {X 0,Y 168.49,Z 1117.216,A -85,B 0,C 180,E1 35769.33,E2 35769.33} C_VEL
LIN {X 0,Y 172.342,Z 1114.043,A -85,B 0,C 180,E1 35769.51,E2 35769.51} C_VEL
LIN {X 0,Y 174.262,Z 1112.118,A -85,B 0,C 180,E1 35773.951,E2 35773.951} C_VEL
LIN {X 0,Y 177.15,Z 1110.924,A -85,B 0,C 180,E1 35783.343,E2 35783.343} C_VEL
LIN {X 0,Y 179.28,Z 1111.465,A -85,B 0,C 180,E1 35789.625,E2 35789.625} C_VEL
LIN {X 0,Y 182.226,Z 1114.208,A -85,B 0,C 180,E1 35797.848,E2 35797.848} C_VEL
LIN {X 0,Y 182.746,Z 1114.947,A -85,B 0,C 180,E1 35799.308,E2 35799.308} C_VEL
LIN {X 0,Y 181.796,Z 1116.816,A -85,B 0,C 180,E1 35800.584,E2 35800.584} C_VEL
LIN {X 0,Y 141.08,Z 1146.842,A -85,B 0,C 180,E1 35801.989,E2 35801.989} C_VEL
LIN {X 0,Y 101.171,Z 1170.009,A -85,B 0,C 180,E1 35804.299,E2 35804.299} C_VEL
LIN {X 0,Y 61.697,Z 1187.326,A -85,B 0,C 180,E1 35808.712,E2 35808.712} C_VEL
LIN {X 0,Y 21.736,Z 1199.785,A -85,B 0,C 180,E1 35825.534,E2 35825.534} C_VEL
LIN {X 0,Y 7.342,Z 1203.954,A -85,B 0,C 180,E1 35909.518,E2 35909.518} C_VEL
LIN {X 0,Y 8.526,Z 1203.88,A -85,B 0,C 180,E1 35969.608,E2 35969.608} C_VEL
LIN {X 0,Y 7.96,Z 1200.101,A -85,B 0,C 180,E1 36080.575,E2 36080.575} C_VEL
LIN {X 0,Y 18.701,Z 1196.384,A -85,B 0,C 180,E1 36111.716,E2 36111.716} C_VEL
LIN {X 0,Y 38.72,Z 1189.496,A -85,B 0,C 180,E1 36126.319,E2 36126.319} C_VEL
LIN {X 0,Y 83.154,Z 1170.644,A -85,B 0,C 180,E1 36128.689,E2 36128.689} C_VEL
LIN {X 0,Y 129.747,Z 1144.485,A -85,B 0,C 180,E1 36130.704,E2 36130.704} C_VEL
LIN {X 0,Y 165.769,Z 1119.079,A -85,B 0,C 180,E1 36131.938,E2 36131.938} C_VEL
LIN {X 0,Y 167.627,Z 1117.563,A -85,B 0,C 180,E1 36132.604,E2 36132.604} C_VEL
LIN {X 0,Y 170.782,Z 1115.927,A -85,B 0,C 180,E1 36142.813,E2 36142.813} C_VEL
LIN {X 0,Y 173.439,Z 1116.77,A -85,B 0,C 180,E1 36150.643,E2 36150.643} C_VEL
LIN {X 0,Y 176.139,Z 1119.24,A -85,B 0,C 180,E1 36157.993,E2 36157.993} C_VEL
LIN {X 0,Y 139.802,Z 1145.682,A -85,B 0,C 180,E1 36158.855,E2 36158.855} C_VEL
LIN {X 0,Y 96.511,Z 1170.368,A -85,B 0,C 180,E1 36160.058,E2 36160.058} C_VEL
LIN {X 0,Y 52.117,Z 1188.713,A -85,B 0,C 180,E1 36162.054,E2 36162.054} C_VEL
LIN {X 0,Y 15.693,Z 1198.993,A -85,B 0,C 180,E1 36165.204,E2 36165.204} C_VEL
LIN {X 0,Y 7.886,Z 1200.645,A -85,B 0,C 180,E1 36165.001,E2 36165.001} C_VEL
LIN {X 0,Y 6.131,Z 1200.642,A -85,B 0,C 180,E1 36147.851,E2 36147.851} C_VEL
LIN {X 0,Y 37.464,Z 1189.945,A -85,B 0,C 180,E1 36126.246,E2 36126.246} C_VEL
LIN {X 0,Y 38.72,Z 1189.496,A -85,B 0,C 180,E1 36126.319,E2 36126.319} C_VEL
LIN {X 0,Y 46.816,Z 1186.537,A -85,B 0,C 180,E1 36128.299,E2 36128.299} C_VEL
LIN {X 0,Y 68.611,Z 1177.693,A -85,B 0,C 180,E1 36134.437,E2 36134.437} C_VEL
LIN {X 0,Y 70.623,Z 1176.77,A -85,B 0,C 180,E1 36134.422,E2 36134.422} C_VEL
LIN {X 0,Y 114.937,Z 1153.764,A -85,B 0,C 180,E1 36134.055,E2 36134.055} C_VEL
LIN {X 0,Y 160.552,Z 1122.949,A -85,B 0,C 180,E1 36134.58,E2 36134.58} C_VEL
LIN {X 0,Y 162.02,Z 1121.858,A -85,B 0,C 180,E1 36134.75,E2 36134.75} C_VEL
LIN {X 0,Y 165.33,Z 1121.11,A -85,B 0,C 180,E1 36145.38,E2 36145.38} C_VEL
LIN {X 0,Y 168.891,Z 1123.029,A -85,B 0,C 180,E1 36155.334,E2 36155.334} C_VEL
LIN {X 0,Y 162.172,Z 1128.448,A -85,B 0,C 180,E1 36155.665,E2 36155.665} C_VEL
LIN {X 0,Y 119.564,Z 1156.307,A -85,B 0,C 180,E1 36155.617,E2 36155.617} C_VEL
LIN {X 0,Y 79.897,Z 1176.32,A -85,B 0,C 180,E1 36155.086,E2 36155.086} C_VEL
LIN {X 0,Y 37.183,Z 1191.846,A -85,B 0,C 180,E1 36151.128,E2 36151.128} C_VEL
LIN {X 0,Y 28.921,Z 1194.214,A -85,B 0,C 180,E1 36148.516,E2 36148.516} C_VEL
LIN {X 0,Y 25.998,Z 1194.879,A -85,B 0,C 180,E1 36144.48,E2 36144.48} C_VEL
LIN {X 0,Y 60.535,Z 1181.348,A -85,B 0,C 180,E1 36134.989,E2 36134.989} C_VEL
LIN {X 0,Y 70.623,Z 1176.77,A -85,B 0,C 180,E1 36134.422,E2 36134.422} C_VEL
LIN {X 0,Y 78.546,Z 1173.243,A -85,B 0,C 180,E1 36135.082,E2 36135.082} C_VEL
LIN {X 0,Y 99.829,Z 1162.727,A -85,B 0,C 180,E1 36138.474,E2 36138.474} C_VEL
LIN {X 0,Y 101.752,Z 1161.634,A -85,B 0,C 180,E1 36138.44,E2 36138.44} C_VEL
LIN {X 0,Y 146.771,Z 1133.382,A -85,B 0,C 180,E1 36137.473,E2 36137.473} C_VEL
LIN {X 0,Y 156.393,Z 1126.237,A -85,B 0,C 180,E1 36137.448,E2 36137.448} C_VEL
LIN {X 0,Y 159.951,Z 1126.346,A -85,B 0,C 180,E1 36148.278,E2 36148.278} C_VEL
LIN {X 0,Y 161.612,Z 1127.22,A -85,B 0,C 180,E1 36152.7,E2 36152.7} C_VEL
LIN {X 0,Y 124.886,Z 1151.695,A -85,B 0,C 180,E1 36152.091,E2 36152.091} C_VEL
LIN {X 0,Y 83.069,Z 1173.411,A -85,B 0,C 180,E1 36149.858,E2 36149.858} C_VEL
LIN {X 0,Y 52.062,Z 1185.709,A -85,B 0,C 180,E1 36144.525,E2 36144.525} C_VEL
LIN {X 0,Y 94.822,Z 1165.473,A -85,B 0,C 180,E1 36138.788,E2 36138.788} C_VEL
LIN {X 0,Y 101.752,Z 1161.634,A -85,B 0,C 180,E1 36138.44,E2 36138.44} C_VEL
LIN {X 0,Y 116.88,Z 1153.185,A -85,B 0,C 180,E1 36139.832,E2 36139.832} C_VEL
LIN {X 0,Y 131.744,Z 1144.141,A -85,B 0,C 180,E1 36141.084,E2 36141.084} C_VEL
LIN {X 0,Y 149.349,Z 1131.927,A -85,B 0,C 180,E1 36140.48,E2 36140.48} C_VEL
LIN {X 0,Y 151.092,Z 1130.698,A -85,B 0,C 180,E1 36140.876,E2 36140.876} C_VEL
LIN {X 0,Y 153.993,Z 1131.267,A -85,B 0,C 180,E1 36149.704,E2 36149.704} C_VEL
LIN {X 0,Y 115.128,Z 1156.095,A -85,B 0,C 180,E1 36147.884,E2 36147.884} C_VEL
LIN {X 0,Y 90.156,Z 1168.994,A -85,B 0,C 180,E1 36145.455,E2 36145.455} C_VEL
LIN {X 0,Y 88.502,Z 1169.585,A -85,B 0,C 180,E1 36144.35,E2 36144.35} C_VEL
LIN {X 0,Y 131.744,Z 1144.141,A -85,B 0,C 180,E1 36141.084,E2 36141.084} C_VEL
LIN {X 0,Y 135.901,Z 1141.654,A -85,B 0,C 180,E1 36142.613,E2 36142.613} C_VEL
LIN {X 0,Y 140.123,Z 1139.143,A -85,B 0,C 180,E1 36144.021,E2 36144.021} C_VEL
LIN {X 0,Y 145.48,Z 1135.46,A -85,B 0,C 180,E1 36143.724,E2 36143.724} C_VEL
LIN {X 0,Y 146.256,Z 1135.542,A -85,B 0,C 180,E1 36145.786,E2 36145.786} C_VEL
LIN {X 0,Y 145.132,Z 1136.53,A -85,B 0,C 180,E1 36146.444,E2 36146.444} C_VEL
LIN {X 0,Y 128.769,Z 1147.097,A -85,B 0,C 180,E1 36145.275,E2 36145.275} C_VEL
LIN {X 0,Y 130.436,Z 1145.836,A -85,B 0,C 180,E1 36144.608,E2 36144.608} C_VEL
LIN {X 0,Y 140.123,Z 1139.143,A -85,B 0,C 180,E1 36144.021,E2 36144.021} C_VEL
LIN {X 0,Y 143.216,Z 1140.794,A -85,B 0,C 180,E1 36143.831,E2 36143.831} C_VEL
LIN {X 0,Y 143.216,Z 1292,A -85,B 0,C 180,E1 36143.831,E2 36143.831} C_VEL
LIN {X 0,Y 143.216,Z 1292,A -85,B 0,C 180,E1 36143.831,E2 36143.831}

QRS_NEXT_CUT()
PTP {E1 36177.224,E2 36177.224}
PTP {X 0,Y 759.882,A -85,B 0,C 180,E1 36177.224,E2 36177.224,E3 0,E4 0,E5 0,E6 0}
QRS_SPEED_INIT()
LIN {X 0,Y 759.882,Z 1292,A -85,B 0,C 180,E1 36177.224,E2 36177.224,E3 0,E4 0,E5 0,E6 0} C_VEL
LIN {X 0,Y 759.882,Z 336.644,A -85,B 0,C 180,E1 36177.224,E2 36177.224} C_VEL
LIN {X 0,Y 759.882,Z 328.565,A -85,B 0,C 180,E1 36177.224,E2 36177.224} C_VEL
LIN {X 0,Y 759.896,Z 326.565,A -85,B 0,C 180,E1 36177.073,E2 36177.073} C_VEL
LIN {X 0,Y 759.908,Z 326.577,A -85,B 0,C 180,E1 36174.033,E2 36174.033} C_VEL
LIN {X 0,Y 759.866,Z 326.57,A -85,B 0,C 180,E1 36171.296,E2 36171.296} C_VEL
LIN {X 0,Y 759.914,Z 326.566,A -85,B 0,C 180,E1 36168.54,E2 36168.54} C_VEL
LIN {X 0,Y 759.882,Z 326.575,A -85,B 0,C 180,E1 36165.6,E2 36165.6} C_VEL
LIN {X 0,Y 759.865,Z 326.569,A -85,B 0,C 180,E1 36162.936,E2 36162.936} C_VEL
LIN {X 0,Y 759.911,Z 326.568,A -85,B 0,C 180,E1 36160.183,E2 36160.183} C_VEL
LIN {X 0,Y 759.873,Z 326.574,A -85,B 0,C 180,E1 36157.281,E2 36157.281} C_VEL
LIN {X 0,Y 759.866,Z 326.569,A -85,B 0,C 180,E1 36154.597,E2 36154.597} C_VEL
LIN {X 0,Y 759.91,Z 326.571,A -85,B 0,C 180,E1 36151.811,E2 36151.811} C_VEL
LIN {X 0,Y 759.869,Z 326.574,A -85,B 0,C 180,E1 36149.035,E2 36149.035} C_VEL
LIN {X 0,Y 759.858,Z 326.57,A -85,B 0,C 180,E1 36146.403,E2 36146.403} C_VEL
LIN {X 0,Y 759.912,Z 326.57,A -85,B 0,C 180,E1 36143.599,E2 36143.599} C_VEL
LIN {X 0,Y 759.867,Z 326.574,A -85,B 0,C 180,E1 36140.809,E2 36140.809} C_VEL
LIN {X 0,Y 759.851,Z 326.571,A -85,B 0,C 180,E1 36138.252,E2 36138.252} C_VEL
LIN {X 0,Y 759.915,Z 326.568,A -85,B 0,C 180,E1 36135.467,E2 36135.467} C_VEL
LIN {X 0,Y 759.862,Z 326.575,A -85,B 0,C 180,E1 36132.559,E2 36132.559} C_VEL
LIN {X 0,Y 759.846,Z 326.572,A -85,B 0,C 180,E1 36130.016,E2 36130.016} C_VEL
LIN {X 0,Y 759.896,Z 326.568,A -85,B 0,C 180,E1 36127.367,E2 36127.367} C_VEL
LIN {X 0,Y 759.867,Z 326.575,A -85,B 0,C 180,E1 36124.406,E2 36124.406} C_VEL
LIN {X 0,Y 759.84,Z 326.573,A -85,B 0,C 180,E1 36121.921,E2 36121.921} C_VEL
LIN {X 0,Y 759.85,Z 326.571,A -85,B 0,C 180,E1 36119.481,E2 36119.481} C_VEL
LIN {X 0,Y 759.916,Z 326.574,A -85,B 0,C 180,E1 36116.659,E2 36116.659} C_VEL
LIN {X 0,Y 759.845,Z 326.574,A -85,B 0,C 180,E1 36113.91,E2 36113.91} C_VEL
LIN {X 0,Y 759.834,Z 326.573,A -85,B 0,C 180,E1 36111.507,E2 36111.507} C_VEL
LIN {X 0,Y 759.855,Z 326.571,A -85,B 0,C 180,E1 36109.047,E2 36109.047} C_VEL
LIN {X 0,Y 759.896,Z 326.577,A -85,B 0,C 180,E1 36106.119,E2 36106.119} C_VEL
LIN {X 0,Y 759.836,Z 326.575,A -85,B 0,C 180,E1 36103.546,E2 36103.546} C_VEL
LIN {X 0,Y 759.827,Z 326.574,A -85,B 0,C 180,E1 36101.231,E2 36101.231} C_VEL
LIN {X 0,Y 759.837,Z 326.573,A -85,B 0,C 180,E1 36098.857,E2 36098.857} C_VEL
LIN {X 0,Y 759.917,Z 326.575,A -85,B 0,C 180,E1 36096.042,E2 36096.042} C_VEL
LIN {X 0,Y 759.835,Z 326.576,A -85,B 0,C 180,E1 36093.319,E2 36093.319} C_VEL
LIN {X 0,Y 759.821,Z 326.575,A -85,B 0,C 180,E1 36090.98,E2 36090.98} C_VEL
LIN {X 0,Y 759.822,Z 326.575,A -85,B 0,C 180,E1 36088.718,E2 36088.718} C_VEL
LIN {X 0,Y 759.856,Z 326.573,A -85,B 0,C 180,E1 36086.228,E2 36086.228} C_VEL
LIN {X 0,Y 759.847,Z 326.576,A -85,B 0,C 180,E1 36083.199,E2 36083.199} C_VEL
LIN {X 0,Y 759.82,Z 326.576,A -85,B 0,C 180,E1 36080.838,E2 36080.838} C_VEL
LIN {X 0,Y 759.813,Z 326.576,A -85,B 0,C 180,E1 36078.616,E2 36078.616} C_VEL
LIN {X 0,Y 759.811,Z 326.576,A -85,B 0,C 180,E1 36076.453,E2 36076.453} C_VEL
LIN {X 0,Y 759.815,Z 326.573,A -85,B 0,C 180,E1 36074.193,E2 36074.193} C_VEL
LIN {X 0,Y 759.861,Z 326.576,A -85,B 0,C 180,E1 36071.67,E2 36071.67} C_VEL
LIN {X 0,Y 759.831,Z 326.578,A -85,B 0,C 180,E1 36068.7,E2 36068.7} C_VEL
LIN {X 0,Y 759.807,Z 326.571,A -85,B 0,C 180,E1 36066.336,E2 36066.336} C_VEL
LIN {X 0,Y 759.877,Z 326.745,A -85,B 0,C 180,E1 36065.376,E2 36065.376} C_VEL
LIN {X 0,Y 759.896,Z 327.871,A -85,B 0,C 180,E1 36065.266,E2 36065.266} C_VEL
LIN {X 0,Y 759.919,Z 527.585,A -85,B 0,C 180,E1 36062.876,E2 36062.876} C_VEL
LIN {X 0,Y 759.912,Z 755.386,A -85,B 0,C 180,E1 36060.229,E2 36060.229} C_VEL
LIN {X 0,Y 759.916,Z 781.752,A -85,B 0,C 180,E1 36059.781,E2 36059.781} C_VEL
LIN {X 0,Y 759.919,Z 807.659,A -85,B 0,C 180,E1 36059.192,E2 36059.192} C_VEL
LIN {X 0,Y 759.917,Z 829.46,A -85,B 0,C 180,E1 36058.576,E2 36058.576} C_VEL
LIN {X 0,Y 759.919,Z 848.555,A -85,B 0,C 180,E1 36057.952,E2 36057.952} C_VEL
LIN {X 0,Y 759.919,Z 868.109,A -85,B 0,C 180,E1 36057.224,E2 36057.224} C_VEL
LIN {X 0,Y 759.913,Z 887.144,A -85,B 0,C 180,E1 36056.426,E2 36056.426} C_VEL
LIN {X 0,Y 759.911,Z 905.982,A -85,B 0,C 180,E1 36055.543,E2 36055.543} C_VEL
LIN {X 0,Y 759.907,Z 925.437,A -85,B 0,C 180,E1 36054.531,E2 36054.531} C_VEL
LIN {X 0,Y 759.917,Z 948.716,A -85,B 0,C 180,E1 36053.178,E2 36053.178} C_VEL
LIN {X 0,Y 759.898,Z 969.618,A -85,B 0,C 180,E1 36051.799,E2 36051.799} C_VEL
LIN {X 0,Y 759.918,Z 987.518,A -85,B 0,C 180,E1 36050.496,E2 36050.496} C_VEL
LIN {X 0,Y 759.901,Z 1007.814,A -85,B 0,C 180,E1 36048.86,E2 36048.86} C_VEL
LIN {X 0,Y 759.901,Z 1025.109,A -85,B 0,C 180,E1 36047.292,E2 36047.292} C_VEL
LIN {X 0,Y 759.883,Z 1039.872,A -85,B 0,C 180,E1 36045.819,E2 36045.819} C_VEL
LIN {X 0,Y 759.898,Z 1056.555,A -85,B 0,C 180,E1 36043.967,E2 36043.967} C_VEL
LIN {X 0,Y 759.907,Z 1070.472,A -85,B 0,C 180,E1 36042.202,E2 36042.202} C_VEL
LIN {X 0,Y 759.885,Z 1081.472,A -85,B 0,C 180,E1 36040.643,E2 36040.643} C_VEL
LIN {X 0,Y 759.916,Z 1091.362,A -85,B 0,C 180,E1 36039.07,E2 36039.07} C_VEL
LIN {X 0,Y 759.878,Z 1100.905,A -85,B 0,C 180,E1 36037.345,E2 36037.345} C_VEL
LIN {X 0,Y 759.881,Z 1110.504,A -85,B 0,C 180,E1 36035.286,E2 36035.286} C_VEL
LIN {X 0,Y 759.917,Z 1117.136,A -85,B 0,C 180,E1 36033.548,E2 36033.548} C_VEL
LIN {X 0,Y 759.906,Z 1123.069,A -85,B 0,C 180,E1 36031.645,E2 36031.645} C_VEL
LIN {X 0,Y 759.905,Z 1127.767,A -85,B 0,C 180,E1 36029.566,E2 36029.566} C_VEL
LIN {X 0,Y 759.902,Z 1130.468,A -85,B 0,C 180,E1 36027.677,E2 36027.677} C_VEL
LIN {X 0,Y 759.912,Z 1131.743,A -85,B 0,C 180,E1 36025.843,E2 36025.843} C_VEL
LIN {X 0,Y 759.883,Z 1131.793,A -85,B 0,C 180,E1 36024.235,E2 36024.235} C_VEL
LIN {X 0,Y 759.864,Z 1130.866,A -85,B 0,C 180,E1 36022.678,E2 36022.678} C_VEL
LIN {X 0,Y 759.906,Z 1128.828,A -85,B 0,C 180,E1 36020.971,E2 36020.971} C_VEL
LIN {X 0,Y 759.904,Z 1124.718,A -85,B 0,C 180,E1 36018.906,E2 36018.906} C_VEL
LIN {X 0,Y 759.879,Z 1119.232,A -85,B 0,C 180,E1 36016.985,E2 36016.985} C_VEL
LIN {X 0,Y 759.911,Z 1113.037,A -85,B 0,C 180,E1 36015.258,E2 36015.258} C_VEL
LIN {X 0,Y 759.912,Z 1106.02,A -85,B 0,C 180,E1 36013.623,E2 36013.623} C_VEL
LIN {X 0,Y 759.909,Z 1098.306,A -85,B 0,C 180,E1 36012.076,E2 36012.076} C_VEL
LIN {X 0,Y 759.882,Z 1089.564,A -85,B 0,C 180,E1 36010.539,E2 36010.539} C_VEL
LIN {X 0,Y 759.887,Z 1078.225,A -85,B 0,C 180,E1 36008.78,E2 36008.78} C_VEL
LIN {X 0,Y 759.897,Z 1063.51,A -85,B 0,C 180,E1 36006.801,E2 36006.801} C_VEL
LIN {X 0,Y 759.914,Z 1050.792,A -85,B 0,C 180,E1 36005.285,E2 36005.285} C_VEL
LIN {X 0,Y 759.886,Z 1037.521,A -85,B 0,C 180,E1 36003.848,E2 36003.848} C_VEL
LIN {X 0,Y 759.91,Z 1022.173,A -85,B 0,C 180,E1 36002.338,E2 36002.338} C_VEL
LIN {X 0,Y 759.908,Z 1002.468,A -85,B 0,C 180,E1 36000.603,E2 36000.603} C_VEL
LIN {X 0,Y 759.915,Z 985.291,A -85,B 0,C 180,E1 35999.246,E2 35999.246} C_VEL
LIN {X 0,Y 759.898,Z 966.429,A -85,B 0,C 180,E1 35997.889,E2 35997.889} C_VEL
LIN {X 0,Y 759.902,Z 942.847,A -85,B 0,C 180,E1 35996.379,E2 35996.379} C_VEL
LIN {X 0,Y 759.912,Z 923.654,A -85,B 0,C 180,E1 35995.283,E2 35995.283} C_VEL
LIN {X 0,Y 759.912,Z 905.359,A -85,B 0,C 180,E1 35994.337,E2 35994.337} C_VEL
LIN {X 0,Y 759.913,Z 886.699,A -85,B 0,C 180,E1 35993.465,E2 35993.465} C_VEL
LIN {X 0,Y 759.919,Z 866.692,A -85,B 0,C 180,E1 35992.629,E2 35992.629} C_VEL
LIN {X 0,Y 759.914,Z 843.876,A -85,B 0,C 180,E1 35991.792,E2 35991.792} C_VEL
LIN {X 0,Y 759.911,Z 815.156,A -85,B 0,C 180,E1 35990.915,E2 35990.915} C_VEL
LIN {X 0,Y 759.911,Z 790.166,A -85,B 0,C 180,E1 35990.304,E2 35990.304} C_VEL
LIN {X 0,Y 759.91,Z 763.464,A -85,B 0,C 180,E1 35989.802,E2 35989.802} C_VEL
LIN {X 0,Y 759.913,Z 734.476,A -85,B 0,C 180,E1 35989.423,E2 35989.423} C_VEL
LIN {X 0,Y 759.918,Z 504.732,A -85,B 0,C 180,E1 35986.765,E2 35986.765} C_VEL
LIN {X 0,Y 759.916,Z 327.648,A -85,B 0,C 180,E1 35984.635,E2 35984.635} C_VEL
LIN {X 0,Y 759.918,Z 326.656,A -85,B 0,C 180,E1 35984.508,E2 35984.508} C_VEL
LIN {X 0,Y 759.847,Z 326.573,A -85,B 0,C 180,E1 35981.818,E2 35981.818} C_VEL
LIN {X 0,Y 759.85,Z 326.571,A -85,B 0,C 180,E1 35979.324,E2 35979.324} C_VEL
LIN {X 0,Y 759.914,Z 326.575,A -85,B 0,C 180,E1 35976.586,E2 35976.586} C_VEL
LIN {X 0,Y 759.873,Z 326.569,A -85,B 0,C 180,E1 35973.76,E2 35973.76} C_VEL
LIN {X 0,Y 759.874,Z 326.574,A -85,B 0,C 180,E1 35971.049,E2 35971.049} C_VEL
LIN {X 0,Y 759.906,Z 326.57,A -85,B 0,C 180,E1 35968.211,E2 35968.211} C_VEL
LIN {X 0,Y 759.879,Z 326.569,A -85,B 0,C 180,E1 35965.449,E2 35965.449} C_VEL
LIN {X 0,Y 759.914,Z 326.577,A -85,B 0,C 180,E1 35962.629,E2 35962.629} C_VEL
LIN {X 0,Y 759.908,Z 326.564,A -85,B 0,C 180,E1 35959.557,E2 35959.557} C_VEL
LIN {X 0,Y 759.894,Z 326.753,A -85,B 0,C 180,E1 35956.825,E2 35956.825} C_VEL
LIN {X 0,Y 759.91,Z 329.397,A -85,B 0,C 180,E1 35956.619,E2 35956.619} C_VEL
LIN {X 0,Y 759.901,Z 370.607,A -85,B 0,C 180,E1 35954.147,E2 35954.147} C_VEL
LIN {X 0,Y 759.909,Z 415.113,A -85,B 0,C 180,E1 35951.588,E2 35951.588} C_VEL
LIN {X 0,Y 759.876,Z 427.188,A -85,B 0,C 180,E1 35950.929,E2 35950.929} C_VEL
LIN {X 0,Y 759.918,Z 624.369,A -85,B 0,C 180,E1 35948.549,E2 35948.549} C_VEL
LIN {X 0,Y 759.908,Z 847.281,A -85,B 0,C 180,E1 35945.956,E2 35945.956} C_VEL
LIN {X 0,Y 759.915,Z 906.046,A -85,B 0,C 180,E1 35945.264,E2 35945.264} C_VEL
LIN {X 0,Y 759.908,Z 932.687,A -85,B 0,C 180,E1 35944.808,E2 35944.808} C_VEL
LIN {X 0,Y 759.909,Z 959.805,A -85,B 0,C 180,E1 35944.183,E2 35944.183} C_VEL
LIN {X 0,Y 759.91,Z 981.822,A -85,B 0,C 180,E1 35943.547,E2 35943.547} C_VEL
LIN {X 0,Y 759.92,Z 999.562,A -85,B 0,C 180,E1 35942.961,E2 35942.961} C_VEL
LIN {X 0,Y 759.918,Z 1017.582,A -85,B 0,C 180,E1 35942.29,E2 35942.29} C_VEL
LIN {X 0,Y 759.913,Z 1036.679,A -85,B 0,C 180,E1 35941.491,E2 35941.491} C_VEL
LIN {X 0,Y 759.91,Z 1055.512,A -85,B 0,C 180,E1 35940.611,E2 35940.611} C_VEL
LIN {X 0,Y 759.911,Z 1074.021,A -85,B 0,C 180,E1 35939.652,E2 35939.652} C_VEL
LIN {X 0,Y 759.906,Z 1094.427,A -85,B 0,C 180,E1 35938.482,E2 35938.482} C_VEL
LIN {X 0,Y 759.913,Z 1117.413,A -85,B 0,C 180,E1 35936.997,E2 35936.997} C_VEL
LIN {X 0,Y 759.904,Z 1134.945,A -85,B 0,C 180,E1 35935.735,E2 35935.735} C_VEL
LIN {X 0,Y 759.9,Z 1152.34,A -85,B 0,C 180,E1 35934.362,E2 35934.362} C_VEL
LIN {X 0,Y 759.915,Z 1173.1,A -85,B 0,C 180,E1 35932.528,E2 35932.528} C_VEL
LIN {X 0,Y 759.902,Z 1188.05,A -85,B 0,C 180,E1 35931.052,E2 35931.052} C_VEL
LIN {X 0,Y 759.884,Z 1201.563,A -85,B 0,C 180,E1 35929.584,E2 35929.584} C_VEL
LIN {X 0,Y 759.897,Z 1216.583,A -85,B 0,C 180,E1 35927.774,E2 35927.774} C_VEL
LIN {X 0,Y 759.882,Z 1229.642,A -85,B 0,C 180,E1 35925.962,E2 35925.962} C_VEL
LIN {X 0,Y 759.915,Z 1239.658,A -85,B 0,C 180,E1 35924.399,E2 35924.399} C_VEL
LIN {X 0,Y 759.906,Z 1248.544,A -85,B 0,C 180,E1 35922.834,E2 35922.834} C_VEL
LIN {X 0,Y 759.911,Z 1256.141,A -85,B 0,C 180,E1 35921.306,E2 35921.306} C_VEL
LIN {X 0,Y 759.889,Z 1262.842,A -85,B 0,C 180,E1 35919.746,E2 35919.746} C_VEL
LIN {X 0,Y 759.9,Z 1268.815,A -85,B 0,C 180,E1 35918.094,E2 35918.094} C_VEL
LIN {X 0,Y 759.916,Z 1274.348,A -85,B 0,C 180,E1 35916.194,E2 35916.194} C_VEL
LIN {X 0,Y 759.918,Z 1278.544,A -85,B 0,C 180,E1 35914.155,E2 35914.155} C_VEL
LIN {X 0,Y 759.904,Z 1280.81,A -85,B 0,C 180,E1 35912.338,E2 35912.338} C_VEL
LIN {X 0,Y 759.864,Z 1281.76,A -85,B 0,C 180,E1 35910.829,E2 35910.829} C_VEL
LIN {X 0,Y 759.862,Z 1281.804,A -85,B 0,C 180,E1 35909.321,E2 35909.321} C_VEL
LIN {X 0,Y 759.911,Z 1280.945,A -85,B 0,C 180,E1 35907.813,E2 35907.813} C_VEL
LIN {X 0,Y 759.913,Z 1278.803,A -85,B 0,C 180,E1 35906.001,E2 35906.001} C_VEL
LIN {X 0,Y 759.913,Z 1274.734,A -85,B 0,C 180,E1 35903.958,E2 35903.958} C_VEL
LIN {X 0,Y 759.888,Z 1269.327,A -85,B 0,C 180,E1 35902.059,E2 35902.059} C_VEL
LIN {X 0,Y 759.884,Z 1263.042,A -85,B 0,C 180,E1 35900.304,E2 35900.304} C_VEL
LIN {X 0,Y 759.906,Z 1256.498,A -85,B 0,C 180,E1 35898.771,E2 35898.771} C_VEL
LIN {X 0,Y 759.912,Z 1248.878,A -85,B 0,C 180,E1 35897.229,E2 35897.229} C_VEL
LIN {X 0,Y 759.914,Z 1240.123,A -85,B 0,C 180,E1 35895.678,E2 35895.678} C_VEL
LIN {X 0,Y 759.883,Z 1230.164,A -85,B 0,C 180,E1 35894.116,E2 35894.116} C_VEL
LIN {X 0,Y 759.89,Z 1217.147,A -85,B 0,C 180,E1 35892.302,E2 35892.302} C_VEL
LIN {X 0,Y 759.887,Z 1202.086,A -85,B 0,C 180,E1 35890.475,E2 35890.475} C_VEL
LIN {X 0,Y 759.904,Z 1188.83,A -85,B 0,C 180,E1 35889.029,E2 35889.029} C_VEL
LIN {X 0,Y 759.907,Z 1174.115,A -85,B 0,C 180,E1 35887.569,E2 35887.569} C_VEL
LIN {X 0,Y 759.891,Z 1155.386,A -85,B 0,C 180,E1 35885.886,E2 35885.886} C_VEL
LIN {X 0,Y 759.915,Z 1136.605,A -85,B 0,C 180,E1 35884.391,E2 35884.391} C_VEL
LIN {X 0,Y 759.918,Z 1119.359,A -85,B 0,C 180,E1 35883.139,E2 35883.139} C_VEL
LIN {X 0,Y 759.917,Z 1097.927,A -85,B 0,C 180,E1 35881.727,E2 35881.727} C_VEL
LIN {X 0,Y 759.907,Z 1075.541,A -85,B 0,C 180,E1 35880.43,E2 35880.43} C_VEL
LIN {X 0,Y 759.913,Z 1056.401,A -85,B 0,C 180,E1 35879.433,E2 35879.433} C_VEL
LIN {X 0,Y 759.912,Z 1037.672,A -85,B 0,C 180,E1 35878.553,E2 35878.553} C_VEL
LIN {X 0,Y 759.918,Z 1018.521,A -85,B 0,C 180,E1 35877.748,E2 35877.748} C_VEL
LIN {X 0,Y 759.919,Z 1000.832,A -85,B 0,C 180,E1 35877.084,E2 35877.084} C_VEL
LIN {X 0,Y 759.91,Z 982.49,A -85,B 0,C 180,E1 35876.473,E2 35876.473} C_VEL
LIN {X 0,Y 759.908,Z 960.609,A -85,B 0,C 180,E1 35875.837,E2 35875.837} C_VEL
LIN {X 0,Y 759.908,Z 933.599,A -85,B 0,C 180,E1 35875.211,E2 35875.211} C_VEL
LIN {X 0,Y 759.916,Z 907.412,A -85,B 0,C 180,E1 35874.756,E2 35874.756} C_VEL
LIN {X 0,Y 759.912,Z 857.465,A -85,B 0,C 180,E1 35874.16,E2 35874.16} C_VEL
LIN {X 0,Y 759.92,Z 633.297,A -85,B 0,C 180,E1 35871.557,E2 35871.557} C_VEL
LIN {X 0,Y 759.876,Z 427.97,A -85,B 0,C 180,E1 35869.083,E2 35869.083} C_VEL
LIN {X 0,Y 759.88,Z 425.732,A -85,B 0,C 180,E1 35869.006,E2 35869.006} C_VEL
LIN {X 0,Y 759.901,Z 378.372,A -85,B 0,C 180,E1 35866.307,E2 35866.307} C_VEL
LIN {X 0,Y 759.918,Z 336.191,A -85,B 0,C 180,E1 35863.797,E2 35863.797} C_VEL
LIN {X 0,Y 759.895,Z 326.883,A -85,B 0,C 180,E1 35863.201,E2 35863.201} C_VEL
LIN {X 0,Y 759.904,Z 326.555,A -85,B 0,C 180,E1 35862.251,E2 35862.251} C_VEL
LIN {X 0,Y 759.91,Z 326.577,A -85,B 0,C 180,E1 35859.315,E2 35859.315} C_VEL
LIN {X 0,Y 759.908,Z 326.562,A -85,B 0,C 180,E1 35856.307,E2 35856.307} C_VEL
LIN {X 0,Y 759.906,Z 326.576,A -85,B 0,C 180,E1 35853.329,E2 35853.329} C_VEL
LIN {X 0,Y 759.884,Z 326.569,A -85,B 0,C 180,E1 35850.473,E2 35850.473} C_VEL
LIN {X 0,Y 759.901,Z 326.567,A -85,B 0,C 180,E1 35847.683,E2 35847.683} C_VEL
LIN {X 0,Y 759.898,Z 326.575,A -85,B 0,C 180,E1 35844.783,E2 35844.783} C_VEL
LIN {X 0,Y 759.903,Z 326.564,A -85,B 0,C 180,E1 35841.862,E2 35841.862} C_VEL
LIN {X 0,Y 759.919,Z 326.577,A -85,B 0,C 180,E1 35838.806,E2 35838.806} C_VEL
LIN {X 0,Y 759.88,Z 326.568,A -85,B 0,C 180,E1 35835.963,E2 35835.963} C_VEL
LIN {X 0,Y 759.902,Z 326.568,A -85,B 0,C 180,E1 35833.173,E2 35833.173} C_VEL
LIN {X 0,Y 759.89,Z 326.574,A -85,B 0,C 180,E1 35830.309,E2 35830.309} C_VEL
LIN {X 0,Y 759.891,Z 326.566,A -85,B 0,C 180,E1 35827.485,E2 35827.485} C_VEL
LIN {X 0,Y 759.906,Z 326.573,A -85,B 0,C 180,E1 35824.604,E2 35824.604} C_VEL
LIN {X 0,Y 759.875,Z 326.572,A -85,B 0,C 180,E1 35821.885,E2 35821.885} C_VEL
LIN {X 0,Y 759.902,Z 326.565,A -85,B 0,C 180,E1 35819.095,E2 35819.095} C_VEL
LIN {X 0,Y 759.896,Z 326.565,A -85,B 0,C 180,E1 35817.073,E2 35817.073} C_VEL
LIN {X 0,Y 758.949,Z 326.691,A -85,B 0,C 180,E1 35816.492,E2 35816.492} C_VEL
LIN {X 0,Y 752.502,Z 327.489,A -85,B 0,C 180,E1 35814.867,E2 35814.867} C_VEL
LIN {X 0,Y 751.967,Z 327.56,A -85,B 0,C 180,E1 35814.444,E2 35814.444} C_VEL
LIN {X 0,Y 751.934,Z 327.562,A -85,B 0,C 180,E1 35811.621,E2 35811.621} C_VEL
LIN {X 0,Y 751.948,Z 327.556,A -85,B 0,C 180,E1 35808.883,E2 35808.883} C_VEL
LIN {X 0,Y 751.974,Z 327.566,A -85,B 0,C 180,E1 35805.838,E2 35805.838} C_VEL
LIN {X 0,Y 751.923,Z 327.559,A -85,B 0,C 180,E1 35803.069,E2 35803.069} C_VEL
LIN {X 0,Y 751.978,Z 327.555,A -85,B 0,C 180,E1 35800.288,E2 35800.288} C_VEL
LIN {X 0,Y 751.937,Z 327.563,A -85,B 0,C 180,E1 35797.317,E2 35797.317} C_VEL
LIN {X 0,Y 751.925,Z 327.558,A -85,B 0,C 180,E1 35794.647,E2 35794.647} C_VEL
LIN {X 0,Y 751.972,Z 327.559,A -85,B 0,C 180,E1 35791.832,E2 35791.832} C_VEL
LIN {X 0,Y 751.93,Z 327.563,A -85,B 0,C 180,E1 35789.028,E2 35789.028} C_VEL
LIN {X 0,Y 751.92,Z 327.559,A -85,B 0,C 180,E1 35786.414,E2 35786.414} C_VEL
LIN {X 0,Y 751.974,Z 327.558,A -85,B 0,C 180,E1 35783.627,E2 35783.627} C_VEL
LIN {X 0,Y 751.929,Z 327.564,A -85,B 0,C 180,E1 35780.827,E2 35780.827} C_VEL
LIN {X 0,Y 751.912,Z 327.56,A -85,B 0,C 180,E1 35778.245,E2 35778.245} C_VEL
LIN {X 0,Y 751.977,Z 327.557,A -85,B 0,C 180,E1 35775.455,E2 35775.455} C_VEL
LIN {X 0,Y 751.923,Z 327.563,A -85,B 0,C 180,E1 35772.549,E2 35772.549} C_VEL
LIN {X 0,Y 751.907,Z 327.561,A -85,B 0,C 180,E1 35770.006,E2 35770.006} C_VEL
LIN {X 0,Y 751.961,Z 327.557,A -85,B 0,C 180,E1 35767.329,E2 35767.329} C_VEL
LIN {X 0,Y 751.929,Z 327.565,A -85,B 0,C 180,E1 35764.412,E2 35764.412} C_VEL
LIN {X 0,Y 751.901,Z 327.562,A -85,B 0,C 180,E1 35761.866,E2 35761.866} C_VEL
LIN {X 0,Y 751.92,Z 327.559,A -85,B 0,C 180,E1 35759.385,E2 35759.385} C_VEL
LIN {X 0,Y 751.966,Z 327.566,A -85,B 0,C 180,E1 35756.452,E2 35756.452} C_VEL
LIN {X 0,Y 751.899,Z 327.562,A -85,B 0,C 180,E1 35753.761,E2 35753.761} C_VEL
LIN {X 0,Y 751.899,Z 327.561,A -85,B 0,C 180,E1 35751.369,E2 35751.369} C_VEL
LIN {X 0,Y 751.967,Z 327.559,A -85,B 0,C 180,E1 35748.69,E2 35748.69} C_VEL
LIN {X 0,Y 751.916,Z 327.564,A -85,B 0,C 180,E1 35745.819,E2 35745.819} C_VEL
LIN {X 0,Y 751.891,Z 327.563,A -85,B 0,C 180,E1 35743.379,E2 35743.379} C_VEL
LIN {X 0,Y 751.893,Z 327.563,A -85,B 0,C 180,E1 35741.04,E2 35741.04} C_VEL
LIN {X 0,Y 751.968,Z 327.56,A -85,B 0,C 180,E1 35738.334,E2 35738.334} C_VEL
LIN {X 0,Y 751.9,Z 327.564,A -85,B 0,C 180,E1 35735.418,E2 35735.418} C_VEL
LIN {X 0,Y 751.884,Z 327.564,A -85,B 0,C 180,E1 35733.049,E2 35733.049} C_VEL
LIN {X 0,Y 751.885,Z 327.563,A -85,B 0,C 180,E1 35730.762,E2 35730.762} C_VEL
LIN {X 0,Y 751.924,Z 327.563,A -85,B 0,C 180,E1 35728.247,E2 35728.247} C_VEL
LIN {X 0,Y 751.911,Z 327.566,A -85,B 0,C 180,E1 35725.271,E2 35725.271} C_VEL
LIN {X 0,Y 751.879,Z 327.564,A -85,B 0,C 180,E1 35722.819,E2 35722.819} C_VEL
LIN {X 0,Y 751.876,Z 327.565,A -85,B 0,C 180,E1 35720.586,E2 35720.586} C_VEL
LIN {X 0,Y 751.884,Z 327.564,A -85,B 0,C 180,E1 35718.26,E2 35718.26} C_VEL
LIN {X 0,Y 751.975,Z 327.56,A -85,B 0,C 180,E1 35715.445,E2 35715.445} C_VEL
LIN {X 0,Y 751.881,Z 327.567,A -85,B 0,C 180,E1 35712.67,E2 35712.67} C_VEL
LIN {X 0,Y 751.87,Z 327.561,A -85,B 0,C 180,E1 35710.42,E2 35710.42} C_VEL
LIN {X 0,Y 751.867,Z 327.569,A -85,B 0,C 180,E1 35708.221,E2 35708.221} C_VEL
LIN {X 0,Y 751.873,Z 327.584,A -85,B 0,C 180,E1 35705.988,E2 35705.988} C_VEL
LIN {X 0,Y 751.984,Z 328.181,A -85,B 0,C 180,E1 35705.805,E2 35705.805} C_VEL
LIN {X 0,Y 753.629,Z 331.614,A -85,B 0,C 180,E1 35705.62,E2 35705.62} C_VEL
LIN {X 0,Y 753.647,Z 476.999,A -85,B 0,C 180,E1 35703.853,E2 35703.853} C_VEL
LIN {X 0,Y 753.421,Z 702.207,A -85,B 0,C 180,E1 35701.213,E2 35701.213} C_VEL
LIN {X 0,Y 753.353,Z 757.623,A -85,B 0,C 180,E1 35700.549,E2 35700.549} C_VEL
LIN {X 0,Y 753.286,Z 783.681,A -85,B 0,C 180,E1 35700.094,E2 35700.094} C_VEL
LIN {X 0,Y 753.199,Z 811.29,A -85,B 0,C 180,E1 35699.447,E2 35699.447} C_VEL
LIN {X 0,Y 753.1,Z 835.698,A -85,B 0,C 180,E1 35698.727,E2 35698.727} C_VEL
LIN {X 0,Y 752.975,Z 861.481,A -85,B 0,C 180,E1 35697.826,E2 35697.826} C_VEL
LIN {X 0,Y 752.861,Z 884.548,A -85,B 0,C 180,E1 35696.872,E2 35696.872} C_VEL
LIN {X 0,Y 752.755,Z 905.161,A -85,B 0,C 180,E1 35695.907,E2 35695.907} C_VEL
LIN {X 0,Y 752.665,Z 924.7,A -85,B 0,C 180,E1 35694.885,E2 35694.885} C_VEL
LIN {X 0,Y 752.551,Z 947.376,A -85,B 0,C 180,E1 35693.565,E2 35693.565} C_VEL
LIN {X 0,Y 752.407,Z 969.107,A -85,B 0,C 180,E1 35692.124,E2 35692.124} C_VEL
LIN {X 0,Y 752.344,Z 987.713,A -85,B 0,C 180,E1 35690.757,E2 35690.757} C_VEL
LIN {X 0,Y 752.215,Z 1007.907,A -85,B 0,C 180,E1 35689.112,E2 35689.112} C_VEL
LIN {X 0,Y 752.164,Z 1025.231,A -85,B 0,C 180,E1 35687.523,E2 35687.523} C_VEL
LIN {X 0,Y 752.082,Z 1040.373,A -85,B 0,C 180,E1 35685.994,E2 35685.994} C_VEL
LIN {X 0,Y 752.028,Z 1057.484,A -85,B 0,C 180,E1 35684.058,E2 35684.058} C_VEL
LIN {X 0,Y 752.004,Z 1070.488,A -85,B 0,C 180,E1 35682.386,E2 35682.386} C_VEL
LIN {X 0,Y 751.94,Z 1081.342,A -85,B 0,C 180,E1 35680.833,E2 35680.833} C_VEL
LIN {X 0,Y 751.938,Z 1091.091,A -85,B 0,C 180,E1 35679.269,E2 35679.269} C_VEL
LIN {X 0,Y 751.928,Z 1100.385,A -85,B 0,C 180,E1 35677.578,E2 35677.578} C_VEL
LIN {X 0,Y 751.886,Z 1110.349,A -85,B 0,C 180,E1 35675.438,E2 35675.438} C_VEL
LIN {X 0,Y 751.921,Z 1117.318,A -85,B 0,C 180,E1 35673.586,E2 35673.586} C_VEL
LIN {X 0,Y 751.908,Z 1123.181,A -85,B 0,C 180,E1 35671.673,E2 35671.673} C_VEL
LIN {X 0,Y 751.905,Z 1127.872,A -85,B 0,C 180,E1 35669.562,E2 35669.562} C_VEL
LIN {X 0,Y 751.899,Z 1130.517,A -85,B 0,C 180,E1 35667.653,E2 35667.653} C_VEL
LIN {X 0,Y 751.913,Z 1131.742,A -85,B 0,C 180,E1 35665.86,E2 35665.86} C_VEL
LIN {X 0,Y 751.882,Z 1131.805,A -85,B 0,C 180,E1 35664.263,E2 35664.263} C_VEL
LIN {X 0,Y 751.866,Z 1130.859,A -85,B 0,C 180,E1 35662.643,E2 35662.643} C_VEL
LIN {X 0,Y 751.909,Z 1128.745,A -85,B 0,C 180,E1 35660.879,E2 35660.879} C_VEL
LIN {X 0,Y 751.906,Z 1124.746,A -85,B 0,C 180,E1 35658.853,E2 35658.853} C_VEL
LIN {X 0,Y 751.884,Z 1119.343,A -85,B 0,C 180,E1 35656.932,E2 35656.932} C_VEL
LIN {X 0,Y 751.922,Z 1113.172,A -85,B 0,C 180,E1 35655.187,E2 35655.187} C_VEL
LIN {X 0,Y 751.933,Z 1106.178,A -85,B 0,C 180,E1 35653.535,E2 35653.535} C_VEL
LIN {X 0,Y 751.933,Z 1098.495,A -85,B 0,C 180,E1 35651.973,E2 35651.973} C_VEL
LIN {X 0,Y 751.921,Z 1089.782,A -85,B 0,C 180,E1 35650.419,E2 35650.419} C_VEL
LIN {X 0,Y 751.955,Z 1078.981,A -85,B 0,C 180,E1 35648.719,E2 35648.719} C_VEL
LIN {X 0,Y 752.005,Z 1063.826,A -85,B 0,C 180,E1 35646.643,E2 35646.643} C_VEL
LIN {X 0,Y 752.073,Z 1050.471,A -85,B 0,C 180,E1 35645.034,E2 35645.034} C_VEL
LIN {X 0,Y 752.109,Z 1036.446,A -85,B 0,C 180,E1 35643.506,E2 35643.506} C_VEL
LIN {X 0,Y 752.182,Z 1018.61,A -85,B 0,C 180,E1 35641.752,E2 35641.752} C_VEL
LIN {X 0,Y 752.275,Z 1000.202,A -85,B 0,C 180,E1 35640.152,E2 35640.152} C_VEL
LIN {X 0,Y 752.356,Z 981.858,A -85,B 0,C 180,E1 35638.705,E2 35638.705} C_VEL
LIN {X 0,Y 752.482,Z 958.534,A -85,B 0,C 180,E1 35637.068,E2 35637.068} C_VEL
LIN {X 0,Y 752.575,Z 939.696,A -85,B 0,C 180,E1 35635.886,E2 35635.886} C_VEL
LIN {X 0,Y 752.676,Z 920.2,A -85,B 0,C 180,E1 35634.779,E2 35634.779} C_VEL
LIN {X 0,Y 752.822,Z 896.074,A -85,B 0,C 180,E1 35633.556,E2 35633.556} C_VEL
LIN {X 0,Y 752.937,Z 872.393,A -85,B 0,C 180,E1 35632.522,E2 35632.522} C_VEL
LIN {X 0,Y 753.029,Z 852.426,A -85,B 0,C 180,E1 35631.755,E2 35631.755} C_VEL
LIN {X 0,Y 753.107,Z 833.056,A -85,B 0,C 180,E1 35631.102,E2 35631.102} C_VEL
LIN {X 0,Y 753.203,Z 810.355,A -85,B 0,C 180,E1 35630.439,E2 35630.439} C_VEL
LIN {X 0,Y 753.286,Z 782.998,A -85,B 0,C 180,E1 35629.803,E2 35629.803} C_VEL
LIN {X 0,Y 753.355,Z 756.356,A -85,B 0,C 180,E1 35629.342,E2 35629.342} C_VEL
LIN {X 0,Y 753.483,Z 643.039,A -85,B 0,C 180,E1 35628.012,E2 35628.012} C_VEL
LIN {X 0,Y 753.701,Z 421.723,A -85,B 0,C 180,E1 35625.394,E2 35625.394} C_VEL
LIN {X 0,Y 753.617,Z 331.535,A -85,B 0,C 180,E1 35624.288,E2 35624.288} C_VEL
LIN {X 0,Y 752.024,Z 328.169,A -85,B 0,C 180,E1 35624.104,E2 35624.104} C_VEL
LIN {X 0,Y 751.913,Z 327.592,A -85,B 0,C 180,E1 35623.943,E2 35623.943} C_VEL
LIN {X 0,Y 751.905,Z 327.566,A -85,B 0,C 180,E1 35621.467,E2 35621.467} C_VEL
LIN {X 0,Y 751.974,Z 327.561,A -85,B 0,C 180,E1 35618.764,E2 35618.764} C_VEL
LIN {X 0,Y 751.931,Z 327.559,A -85,B 0,C 180,E1 35615.811,E2 35615.811} C_VEL
LIN {X 0,Y 751.927,Z 327.563,A -85,B 0,C 180,E1 35613.159,E2 35613.159} C_VEL
LIN {X 0,Y 751.969,Z 327.561,A -85,B 0,C 180,E1 35610.353,E2 35610.353} C_VEL
LIN {X 0,Y 751.938,Z 327.558,A -85,B 0,C 180,E1 35607.505,E2 35607.505} C_VEL
LIN {X 0,Y 751.974,Z 327.567,A -85,B 0,C 180,E1 35604.661,E2 35604.661} C_VEL
LIN {X 0,Y 751.965,Z 327.556,A -85,B 0,C 180,E1 35601.613,E2 35601.613} C_VEL
LIN {X 0,Y 751.969,Z 327.542,A -85,B 0,C 180,E1 35598.634,E2 35598.634} C_VEL
LIN {X 0,Y 751.989,Z 327.733,A -85,B 0,C 180,E1 35597.406,E2 35597.406} C_VEL
LIN {X 0,Y 753.152,Z 330.876,A -85,B 0,C 180,E1 35597.073,E2 35597.073} C_VEL
LIN {X 0,Y 753.735,Z 331.85,A -85,B 0,C 180,E1 35596.965,E2 35596.965} C_VEL
LIN {X 0,Y 753.564,Z 373.005,A -85,B 0,C 180,E1 35594.474,E2 35594.474} C_VEL
LIN {X 0,Y 753.397,Z 417.739,A -85,B 0,C 180,E1 35591.879,E2 35591.879} C_VEL
LIN {X 0,Y 753.513,Z 427.665,A -85,B 0,C 180,E1 35591.342,E2 35591.342} C_VEL
LIN {X 0,Y 753.811,Z 431.219,A -85,B 0,C 180,E1 35591.276,E2 35591.276} C_VEL
LIN {X 0,Y 753.629,Z 641.424,A -85,B 0,C 180,E1 35588.726,E2 35588.726} C_VEL
LIN {X 0,Y 753.412,Z 867.655,A -85,B 0,C 180,E1 35586.08,E2 35586.08} C_VEL
LIN {X 0,Y 753.356,Z 909.047,A -85,B 0,C 180,E1 35585.573,E2 35585.573} C_VEL
LIN {X 0,Y 753.271,Z 935.188,A -85,B 0,C 180,E1 35585.107,E2 35585.107} C_VEL
LIN {X 0,Y 753.183,Z 961.948,A -85,B 0,C 180,E1 35584.475,E2 35584.475} C_VEL
LIN {X 0,Y 753.093,Z 986.883,A -85,B 0,C 180,E1 35583.734,E2 35583.734} C_VEL
LIN {X 0,Y 752.955,Z 1014.23,A -85,B 0,C 180,E1 35582.761,E2 35582.761} C_VEL
LIN {X 0,Y 752.856,Z 1035.688,A -85,B 0,C 180,E1 35581.865,E2 35581.865} C_VEL
LIN {X 0,Y 752.755,Z 1054.625,A -85,B 0,C 180,E1 35580.978,E2 35580.978} C_VEL
LIN {X 0,Y 752.662,Z 1074.023,A -85,B 0,C 180,E1 35579.967,E2 35579.967} C_VEL
LIN {X 0,Y 752.557,Z 1095.065,A -85,B 0,C 180,E1 35578.748,E2 35578.748} C_VEL
LIN {X 0,Y 752.424,Z 1117.976,A -85,B 0,C 180,E1 35577.248,E2 35577.248} C_VEL
LIN {X 0,Y 752.331,Z 1135.499,A -85,B 0,C 180,E1 35575.971,E2 35575.971} C_VEL
LIN {X 0,Y 752.261,Z 1153.356,A -85,B 0,C 180,E1 35574.542,E2 35574.542} C_VEL
LIN {X 0,Y 752.174,Z 1173.264,A -85,B 0,C 180,E1 35572.757,E2 35572.757} C_VEL
LIN {X 0,Y 752.104,Z 1188.263,A -85,B 0,C 180,E1 35571.258,E2 35571.258} C_VEL
LIN {X 0,Y 752.036,Z 1202.23,A -85,B 0,C 180,E1 35569.721,E2 35569.721} C_VEL
LIN {X 0,Y 751.983,Z 1218.336,A -85,B 0,C 180,E1 35567.727,E2 35567.727} C_VEL
LIN {X 0,Y 751.948,Z 1230.166,A -85,B 0,C 180,E1 35566.056,E2 35566.056} C_VEL
LIN {X 0,Y 751.961,Z 1240.125,A -85,B 0,C 180,E1 35564.476,E2 35564.476} C_VEL
LIN {X 0,Y 751.927,Z 1248.88,A -85,B 0,C 180,E1 35562.909,E2 35562.909} C_VEL
LIN {X 0,Y 751.928,Z 1256.499,A -85,B 0,C 180,E1 35561.35,E2 35561.35} C_VEL
LIN {X 0,Y 751.888,Z 1263.655,A -85,B 0,C 180,E1 35559.646,E2 35559.646} C_VEL
LIN {X 0,Y 751.89,Z 1271.033,A -85,B 0,C 180,E1 35557.488,E2 35557.488} C_VEL
LIN {X 0,Y 751.907,Z 1276.28,A -85,B 0,C 180,E1 35555.418,E2 35555.418} C_VEL
LIN {X 0,Y 751.908,Z 1279.789,A -85,B 0,C 180,E1 35553.354,E2 35553.354} C_VEL
LIN {X 0,Y 751.884,Z 1281.67,A -85,B 0,C 180,E1 35551.143,E2 35551.143} C_VEL
LIN {X 0,Y 751.865,Z 1281.849,A -85,B 0,C 180,E1 35549.467,E2 35549.467} C_VEL
LIN {X 0,Y 751.913,Z 1281.013,A -85,B 0,C 180,E1 35547.866,E2 35547.866} C_VEL
LIN {X 0,Y 751.912,Z 1278.928,A -85,B 0,C 180,E1 35546.035,E2 35546.035} C_VEL
LIN {X 0,Y 751.917,Z 1274.734,A -85,B 0,C 180,E1 35543.893,E2 35543.893} C_VEL
LIN {X 0,Y 751.898,Z 1269.327,A -85,B 0,C 180,E1 35541.974,E2 35541.974} C_VEL
LIN {X 0,Y 751.906,Z 1263.024,A -85,B 0,C 180,E1 35540.195,E2 35540.195} C_VEL
LIN {X 0,Y 751.928,Z 1256.141,A -85,B 0,C 180,E1 35538.572,E2 35538.572} C_VEL
LIN {X 0,Y 751.919,Z 1248.469,A -85,B 0,C 180,E1 35537.013,E2 35537.013} C_VEL
LIN {X 0,Y 751.959,Z 1239.66,A -85,B 0,C 180,E1 35535.445,E2 35535.445} C_VEL
LIN {X 0,Y 751.959,Z 1228.598,A -85,B 0,C 180,E1 35533.706,E2 35533.706} C_VEL
LIN {X 0,Y 752.024,Z 1213.375,A -85,B 0,C 180,E1 35531.633,E2 35531.633} C_VEL
LIN {X 0,Y 752.04,Z 1200.252,A -85,B 0,C 180,E1 35530.054,E2 35530.054} C_VEL
LIN {X 0,Y 752.116,Z 1186.492,A -85,B 0,C 180,E1 35528.556,E2 35528.556} C_VEL
LIN {X 0,Y 752.193,Z 1168.498,A -85,B 0,C 180,E1 35526.788,E2 35526.788} C_VEL
LIN {X 0,Y 752.281,Z 1150.276,A -85,B 0,C 180,E1 35525.205,E2 35525.205} C_VEL
LIN {X 0,Y 752.332,Z 1133.284,A -85,B 0,C 180,E1 35523.859,E2 35523.859} C_VEL
LIN {X 0,Y 752.476,Z 1111.182,A -85,B 0,C 180,E1 35522.285,E2 35522.285} C_VEL
LIN {X 0,Y 752.573,Z 1090.697,A -85,B 0,C 180,E1 35520.991,E2 35520.991} C_VEL
LIN {X 0,Y 752.668,Z 1072.416,A -85,B 0,C 180,E1 35519.946,E2 35519.946} C_VEL
LIN {X 0,Y 752.762,Z 1052.844,A -85,B 0,C 180,E1 35518.933,E2 35518.933} C_VEL
LIN {X 0,Y 752.91,Z 1028.71,A -85,B 0,C 180,E1 35517.823,E2 35517.823} C_VEL
LIN {X 0,Y 753.022,Z 1004.651,A -85,B 0,C 180,E1 35516.88,E2 35516.88} C_VEL
LIN {X 0,Y 753.101,Z 984.022,A -85,B 0,C 180,E1 35516.177,E2 35516.177} C_VEL
LIN {X 0,Y 753.191,Z 960.817,A -85,B 0,C 180,E1 35515.496,E2 35515.496} C_VEL
LIN {X 0,Y 753.277,Z 933.165,A -85,B 0,C 180,E1 35514.85,E2 35514.85} C_VEL
LIN {X 0,Y 753.357,Z 906.258,A -85,B 0,C 180,E1 35514.386,E2 35514.386} C_VEL
LIN {X 0,Y 753.465,Z 810.565,A -85,B 0,C 180,E1 35513.261,E2 35513.261} C_VEL
LIN {X 0,Y 753.673,Z 590.768,A -85,B 0,C 180,E1 35510.668,E2 35510.668} C_VEL
LIN {X 0,Y 753.739,Z 428.669,A -85,B 0,C 180,E1 35508.687,E2 35508.687} C_VEL
LIN {X 0,Y 753.35,Z 425.9,A -85,B 0,C 180,E1 35508.582,E2 35508.582} C_VEL
LIN {X 0,Y 753.533,Z 378.992,A -85,B 0,C 180,E1 35505.879,E2 35505.879} C_VEL
LIN {X 0,Y 753.724,Z 337.216,A -85,B 0,C 180,E1 35503.367,E2 35503.367} C_VEL
LIN {X 0,Y 753.582,Z 331.491,A -85,B 0,C 180,E1 35503,E2 35503} C_VEL
LIN {X 0,Y 752.002,Z 327.829,A -85,B 0,C 180,E1 35502.615,E2 35502.615} C_VEL
LIN {X 0,Y 751.971,Z 327.544,A -85,B 0,C 180,E1 35501.366,E2 35501.366} C_VEL
LIN {X 0,Y 751.969,Z 327.551,A -85,B 0,C 180,E1 35498.325,E2 35498.325} C_VEL
LIN {X 0,Y 751.972,Z 327.564,A -85,B 0,C 180,E1 35495.246,E2 35495.246} C_VEL
LIN {X 0,Y 751.957,Z 327.556,A -85,B 0,C 180,E1 35492.313,E2 35492.313} C_VEL
LIN {X 0,Y 751.958,Z 327.562,A -85,B 0,C 180,E1 35489.431,E2 35489.431} C_VEL
LIN {X 0,Y 751.949,Z 327.562,A -85,B 0,C 180,E1 35486.675,E2 35486.675} C_VEL
LIN {X 0,Y 751.974,Z 327.552,A -85,B 0,C 180,E1 35483.821,E2 35483.821} C_VEL
LIN {X 0,Y 751.969,Z 327.566,A -85,B 0,C 180,E1 35480.795,E2 35480.795} C_VEL
LIN {X 0,Y 751.95,Z 327.555,A -85,B 0,C 180,E1 35477.889,E2 35477.889} C_VEL
LIN {X 0,Y 751.96,Z 327.56,A -85,B 0,C 180,E1 35475.028,E2 35475.028} C_VEL
LIN {X 0,Y 751.942,Z 327.561,A -85,B 0,C 180,E1 35472.219,E2 35472.219} C_VEL
LIN {X 0,Y 751.968,Z 327.553,A -85,B 0,C 180,E1 35469.383,E2 35469.383} C_VEL
LIN {X 0,Y 751.965,Z 327.564,A -85,B 0,C 180,E1 35466.336,E2 35466.336} C_VEL
LIN {X 0,Y 751.94,Z 327.557,A -85,B 0,C 180,E1 35463.507,E2 35463.507} C_VEL
LIN {X 0,Y 751.965,Z 327.558,A -85,B 0,C 180,E1 35460.686,E2 35460.686} C_VEL
LIN {X 0,Y 751.941,Z 327.563,A -85,B 0,C 180,E1 35457.866,E2 35457.866} C_VEL
LIN {X 0,Y 751.946,Z 327.556,A -85,B 0,C 180,E1 35455.118,E2 35455.118} C_VEL
LIN {X 0,Y 751.967,Z 327.56,A -85,B 0,C 180,E1 35454.444,E2 35454.444} C_VEL
LIN {X 0,Y 750.991,Z 327.692,A -85,B 0,C 180,E1 35453.857,E2 35453.857} C_VEL
LIN {X 0,Y 744.568,Z 328.491,A -85,B 0,C 180,E1 35452.214,E2 35452.214} C_VEL
LIN {X 0,Y 744.007,Z 328.553,A -85,B 0,C 180,E1 35451.787,E2 35451.787} C_VEL
LIN {X 0,Y 743.999,Z 328.546,A -85,B 0,C 180,E1 35448.998,E2 35448.998} C_VEL
LIN {X 0,Y 744.032,Z 328.552,A -85,B 0,C 180,E1 35446.081,E2 35446.081} C_VEL
LIN {X 0,Y 743.987,Z 328.55,A -85,B 0,C 180,E1 35443.285,E2 35443.285} C_VEL
LIN {X 0,Y 744.015,Z 328.545,A -85,B 0,C 180,E1 35440.531,E2 35440.531} C_VEL
LIN {X 0,Y 744.015,Z 328.553,A -85,B 0,C 180,E1 35437.479,E2 35437.479} C_VEL
LIN {X 0,Y 743.982,Z 328.548,A -85,B 0,C 180,E1 35434.753,E2 35434.753} C_VEL
LIN {X 0,Y 744.036,Z 328.546,A -85,B 0,C 180,E1 35431.942,E2 35431.942} C_VEL
LIN {X 0,Y 743.992,Z 328.552,A -85,B 0,C 180,E1 35429.02,E2 35429.02} C_VEL
LIN {X 0,Y 743.983,Z 328.548,A -85,B 0,C 180,E1 35426.377,E2 35426.377} C_VEL
LIN {X 0,Y 744.035,Z 328.548,A -85,B 0,C 180,E1 35423.559,E2 35423.559} C_VEL
LIN {X 0,Y 743.984,Z 328.552,A -85,B 0,C 180,E1 35420.725,E2 35420.725} C_VEL
LIN {X 0,Y 743.979,Z 328.548,A -85,B 0,C 180,E1 35418.121,E2 35418.121} C_VEL
LIN {X 0,Y 744.037,Z 328.551,A -85,B 0,C 180,E1 35415.236,E2 35415.236} C_VEL
LIN {X 0,Y 743.975,Z 328.551,A -85,B 0,C 180,E1 35412.428,E2 35412.428} C_VEL
LIN {X 0,Y 743.975,Z 328.549,A -85,B 0,C 180,E1 35409.872,E2 35409.872} C_VEL
LIN {X 0,Y 744.038,Z 328.548,A -85,B 0,C 180,E1 35407.113,E2 35407.113} C_VEL
LIN {X 0,Y 743.976,Z 328.553,A -85,B 0,C 180,E1 35404.254,E2 35404.254} C_VEL
LIN {X 0,Y 743.966,Z 328.55,A -85,B 0,C 180,E1 35401.706,E2 35401.706} C_VEL
LIN {X 0,Y 744.041,Z 328.546,A -85,B 0,C 180,E1 35398.933,E2 35398.933} C_VEL
LIN {X 0,Y 743.978,Z 328.553,A -85,B 0,C 180,E1 35396.07,E2 35396.07} C_VEL
LIN {X 0,Y 743.958,Z 328.55,A -85,B 0,C 180,E1 35393.563,E2 35393.563} C_VEL
LIN {X 0,Y 743.988,Z 328.549,A -85,B 0,C 180,E1 35391.028,E2 35391.028} C_VEL
LIN {X 0,Y 743.983,Z 328.554,A -85,B 0,C 180,E1 35387.925,E2 35387.925} C_VEL
LIN {X 0,Y 743.953,Z 328.552,A -85,B 0,C 180,E1 35385.433,E2 35385.433} C_VEL
LIN {X 0,Y 743.959,Z 328.551,A -85,B 0,C 180,E1 35383.049,E2 35383.049} C_VEL
LIN {X 0,Y 744.037,Z 328.551,A -85,B 0,C 180,E1 35380.296,E2 35380.296} C_VEL
LIN {X 0,Y 743.964,Z 328.554,A -85,B 0,C 180,E1 35377.491,E2 35377.491} C_VEL
LIN {X 0,Y 743.947,Z 328.552,A -85,B 0,C 180,E1 35375.089,E2 35375.089} C_VEL
LIN {X 0,Y 743.95,Z 328.552,A -85,B 0,C 180,E1 35372.773,E2 35372.773} C_VEL
LIN {X 0,Y 744.041,Z 328.55,A -85,B 0,C 180,E1 35370,E2 35370} C_VEL
LIN {X 0,Y 743.955,Z 328.552,A -85,B 0,C 180,E1 35367.15,E2 35367.15} C_VEL
LIN {X 0,Y 743.942,Z 328.554,A -85,B 0,C 180,E1 35364.834,E2 35364.834} C_VEL
LIN {X 0,Y 743.941,Z 328.551,A -85,B 0,C 180,E1 35362.509,E2 35362.509} C_VEL
LIN {X 0,Y 743.977,Z 328.553,A -85,B 0,C 180,E1 35360.016,E2 35360.016} C_VEL
LIN {X 0,Y 743.96,Z 328.554,A -85,B 0,C 180,E1 35356.951,E2 35356.951} C_VEL
LIN {X 0,Y 743.934,Z 328.542,A -85,B 0,C 180,E1 35354.567,E2 35354.567} C_VEL
LIN {X 0,Y 743.931,Z 328.557,A -85,B 0,C 180,E1 35352.317,E2 35352.317} C_VEL
LIN {X 0,Y 743.938,Z 328.547,A -85,B 0,C 180,E1 35350.039,E2 35350.039} C_VEL
LIN {X 0,Y 744.023,Z 328.539,A -85,B 0,C 180,E1 35347.313,E2 35347.313} C_VEL
LIN {X 0,Y 743.963,Z 328.765,A -85,B 0,C 180,E1 35346.39,E2 35346.39} C_VEL
LIN {X 0,Y 744.284,Z 330.101,A -85,B 0,C 180,E1 35346.264,E2 35346.264} C_VEL
LIN {X 0,Y 746.238,Z 333.238,A -85,B 0,C 180,E1 35346.089,E2 35346.089} C_VEL
LIN {X 0,Y 747.48,Z 334.965,A -85,B 0,C 180,E1 35345.985,E2 35345.985} C_VEL
LIN {X 0,Y 747.701,Z 338.745,A -85,B 0,C 180,E1 35345.923,E2 35345.923} C_VEL
LIN {X 0,Y 747.242,Z 555.036,A -85,B 0,C 180,E1 35343.307,E2 35343.307} C_VEL
LIN {X 0,Y 746.828,Z 756.203,A -85,B 0,C 180,E1 35340.93,E2 35340.93} C_VEL
LIN {X 0,Y 746.696,Z 782.934,A -85,B 0,C 180,E1 35340.466,E2 35340.466} C_VEL
LIN {X 0,Y 746.52,Z 810.142,A -85,B 0,C 180,E1 35339.83,E2 35339.83} C_VEL
LIN {X 0,Y 746.327,Z 834.025,A -85,B 0,C 180,E1 35339.128,E2 35339.128} C_VEL
LIN {X 0,Y 746.146,Z 856.445,A -85,B 0,C 180,E1 35338.357,E2 35338.357} C_VEL
LIN {X 0,Y 745.833,Z 883.599,A -85,B 0,C 180,E1 35337.253,E2 35337.253} C_VEL
LIN {X 0,Y 745.624,Z 904.975,A -85,B 0,C 180,E1 35336.246,E2 35336.246} C_VEL
LIN {X 0,Y 745.431,Z 925.689,A -85,B 0,C 180,E1 35335.151,E2 35335.151} C_VEL
LIN {X 0,Y 745.16,Z 949.775,A -85,B 0,C 180,E1 35333.719,E2 35333.719} C_VEL
LIN {X 0,Y 744.931,Z 969.967,A -85,B 0,C 180,E1 35332.359,E2 35332.359} C_VEL
LIN {X 0,Y 744.778,Z 989.165,A -85,B 0,C 180,E1 35330.927,E2 35330.927} C_VEL
LIN {X 0,Y 744.531,Z 1010.368,A -85,B 0,C 180,E1 35329.155,E2 35329.155} C_VEL
LIN {X 0,Y 744.419,Z 1025.884,A -85,B 0,C 180,E1 35327.707,E2 35327.707} C_VEL
LIN {X 0,Y 744.28,Z 1041.92,A -85,B 0,C 180,E1 35326.061,E2 35326.061} C_VEL
LIN {X 0,Y 744.155,Z 1058.746,A -85,B 0,C 180,E1 35324.108,E2 35324.108} C_VEL
LIN {X 0,Y 744.098,Z 1070.868,A -85,B 0,C 180,E1 35322.525,E2 35322.525} C_VEL
LIN {X 0,Y 744.003,Z 1081.717,A -85,B 0,C 180,E1 35320.95,E2 35320.95} C_VEL
LIN {X 0,Y 743.985,Z 1091.973,A -85,B 0,C 180,E1 35319.275,E2 35319.275} C_VEL
LIN {X 0,Y 743.916,Z 1102.918,A -85,B 0,C 180,E1 35317.218,E2 35317.218} C_VEL
LIN {X 0,Y 743.903,Z 1111.302,A -85,B 0,C 180,E1 35315.308,E2 35315.308} C_VEL
LIN {X 0,Y 743.925,Z 1117.499,A -85,B 0,C 180,E1 35313.625,E2 35313.625} C_VEL
LIN {X 0,Y 743.91,Z 1123.293,A -85,B 0,C 180,E1 35311.701,E2 35311.701} C_VEL
LIN {X 0,Y 743.906,Z 1127.917,A -85,B 0,C 180,E1 35309.585,E2 35309.585} C_VEL
LIN {X 0,Y 743.895,Z 1130.567,A -85,B 0,C 180,E1 35307.628,E2 35307.628} C_VEL
LIN {X 0,Y 743.912,Z 1131.759,A -85,B 0,C 180,E1 35305.816,E2 35305.816} C_VEL
LIN {X 0,Y 743.884,Z 1131.791,A -85,B 0,C 180,E1 35304.203,E2 35304.203} C_VEL
LIN {X 0,Y 743.87,Z 1130.817,A -85,B 0,C 180,E1 35302.567,E2 35302.567} C_VEL
LIN {X 0,Y 743.913,Z 1128.662,A -85,B 0,C 180,E1 35300.784,E2 35300.784} C_VEL
LIN {X 0,Y 743.911,Z 1124.627,A -85,B 0,C 180,E1 35298.738,E2 35298.738} C_VEL
LIN {X 0,Y 743.893,Z 1119.189,A -85,B 0,C 180,E1 35296.798,E2 35296.798} C_VEL
LIN {X 0,Y 743.938,Z 1112.993,A -85,B 0,C 180,E1 35295.035,E2 35295.035} C_VEL
LIN {X 0,Y 743.945,Z 1105.802,A -85,B 0,C 180,E1 35293.328,E2 35293.328} C_VEL
LIN {X 0,Y 743.964,Z 1097.458,A -85,B 0,C 180,E1 35291.631,E2 35291.631} C_VEL
LIN {X 0,Y 744.01,Z 1086.328,A -85,B 0,C 180,E1 35289.671,E2 35289.671} C_VEL
LIN {X 0,Y 744.07,Z 1073.318,A -85,B 0,C 180,E1 35287.723,E2 35287.723} C_VEL
LIN {X 0,Y 744.124,Z 1061.682,A -85,B 0,C 180,E1 35286.171,E2 35286.171} C_VEL
LIN {X 0,Y 744.239,Z 1048.814,A -85,B 0,C 180,E1 35284.624,E2 35284.624} C_VEL
LIN {X 0,Y 744.386,Z 1032.463,A -85,B 0,C 180,E1 35282.849,E2 35282.849} C_VEL
LIN {X 0,Y 744.534,Z 1013.934,A -85,B 0,C 180,E1 35281.077,E2 35281.077} C_VEL
LIN {X 0,Y 744.661,Z 996.112,A -85,B 0,C 180,E1 35279.538,E2 35279.538} C_VEL
LIN {X 0,Y 744.908,Z 974.09,A -85,B 0,C 180,E1 35277.846,E2 35277.846} C_VEL
LIN {X 0,Y 745.105,Z 955.065,A -85,B 0,C 180,E1 35276.538,E2 35276.538} C_VEL
LIN {X 0,Y 745.329,Z 933.358,A -85,B 0,C 180,E1 35275.19,E2 35275.19} C_VEL
LIN {X 0,Y 745.601,Z 909.259,A -85,B 0,C 180,E1 35273.88,E2 35273.88} C_VEL
LIN {X 0,Y 745.807,Z 888.421,A -85,B 0,C 180,E1 35272.876,E2 35272.876} C_VEL
LIN {X 0,Y 746.004,Z 867.612,A -85,B 0,C 180,E1 35271.987,E2 35271.987} C_VEL
LIN {X 0,Y 746.215,Z 843.751,A -85,B 0,C 180,E1 35271.097,E2 35271.097} C_VEL
LIN {X 0,Y 746.459,Z 814.985,A -85,B 0,C 180,E1 35270.21,E2 35270.21} C_VEL
LIN {X 0,Y 746.656,Z 789.208,A -85,B 0,C 180,E1 35269.577,E2 35269.577} C_VEL
LIN {X 0,Y 746.797,Z 762.606,A -85,B 0,C 180,E1 35269.077,E2 35269.077} C_VEL
LIN {X 0,Y 746.909,Z 729.398,A -85,B 0,C 180,E1 35268.648,E2 35268.648} C_VEL
LIN {X 0,Y 747.36,Z 500.22,A -85,B 0,C 180,E1 35265.949,E2 35265.949} C_VEL
LIN {X 0,Y 747.603,Z 335.115,A -85,B 0,C 180,E1 35263.936,E2 35263.936} C_VEL
LIN {X 0,Y 746.421,Z 333.375,A -85,B 0,C 180,E1 35263.835,E2 35263.835} C_VEL
LIN {X 0,Y 744.403,Z 330.348,A -85,B 0,C 180,E1 35263.658,E2 35263.658} C_VEL
LIN {X 0,Y 743.999,Z 328.82,A -85,B 0,C 180,E1 35263.526,E2 35263.526} C_VEL
LIN {X 0,Y 744.025,Z 328.549,A -85,B 0,C 180,E1 35262.319,E2 35262.319} C_VEL
LIN {X 0,Y 743.968,Z 328.538,A -85,B 0,C 180,E1 35259.629,E2 35259.629} C_VEL
LIN {X 0,Y 744,Z 328.556,A -85,B 0,C 180,E1 35257.011,E2 35257.011} C_VEL
LIN {X 0,Y 744.013,Z 328.547,A -85,B 0,C 180,E1 35253.93,E2 35253.93} C_VEL
LIN {X 0,Y 743.989,Z 328.552,A -85,B 0,C 180,E1 35251.193,E2 35251.193} C_VEL
LIN {X 0,Y 744.031,Z 328.553,A -85,B 0,C 180,E1 35248.431,E2 35248.431} C_VEL
LIN {X 0,Y 744.008,Z 328.547,A -85,B 0,C 180,E1 35245.543,E2 35245.543} C_VEL
LIN {X 0,Y 744.029,Z 328.556,A -85,B 0,C 180,E1 35242.692,E2 35242.692} C_VEL
LIN {X 0,Y 744.04,Z 328.541,A -85,B 0,C 180,E1 35239.628,E2 35239.628} C_VEL
LIN {X 0,Y 744.05,Z 328.777,A -85,B 0,C 180,E1 35237.999,E2 35237.999} C_VEL
LIN {X 0,Y 745.278,Z 331.909,A -85,B 0,C 180,E1 35237.662,E2 35237.662} C_VEL
LIN {X 0,Y 746.437,Z 334.008,A -85,B 0,C 180,E1 35237.431,E2 35237.431} C_VEL
LIN {X 0,Y 747.581,Z 336.692,A -85,B 0,C 180,E1 35237.166,E2 35237.166} C_VEL
LIN {X 0,Y 747.219,Z 378.373,A -85,B 0,C 180,E1 35234.629,E2 35234.629} C_VEL
LIN {X 0,Y 746.889,Z 423.912,A -85,B 0,C 180,E1 35231.971,E2 35231.971} C_VEL
LIN {X 0,Y 747.09,Z 428.007,A -85,B 0,C 180,E1 35231.771,E2 35231.771} C_VEL
LIN {X 0,Y 747.782,Z 432.11,A -85,B 0,C 180,E1 35231.672,E2 35231.672} C_VEL
LIN {X 0,Y 747.374,Z 642.34,A -85,B 0,C 180,E1 35229.101,E2 35229.101} C_VEL
LIN {X 0,Y 746.935,Z 868.457,A -85,B 0,C 180,E1 35226.433,E2 35226.433} C_VEL
LIN {X 0,Y 746.823,Z 909.433,A -85,B 0,C 180,E1 35225.926,E2 35225.926} C_VEL
LIN {X 0,Y 746.66,Z 935.865,A -85,B 0,C 180,E1 35225.45,E2 35225.45} C_VEL
LIN {X 0,Y 746.489,Z 962.299,A -85,B 0,C 180,E1 35224.818,E2 35224.818} C_VEL
LIN {X 0,Y 746.298,Z 988.426,A -85,B 0,C 180,E1 35224.034,E2 35224.034} C_VEL
LIN {X 0,Y 746.013,Z 1015.353,A -85,B 0,C 180,E1 35223.059,E2 35223.059} C_VEL
LIN {X 0,Y 745.814,Z 1036.685,A -85,B 0,C 180,E1 35222.157,E2 35222.157} C_VEL
LIN {X 0,Y 745.614,Z 1056.497,A -85,B 0,C 180,E1 35221.214,E2 35221.214} C_VEL
LIN {X 0,Y 745.41,Z 1078.04,A -85,B 0,C 180,E1 35220.066,E2 35220.066} C_VEL
LIN {X 0,Y 745.121,Z 1101.913,A -85,B 0,C 180,E1 35218.624,E2 35218.624} C_VEL
LIN {X 0,Y 744.939,Z 1120.439,A -85,B 0,C 180,E1 35217.368,E2 35217.368} C_VEL
LIN {X 0,Y 744.767,Z 1138.267,A -85,B 0,C 180,E1 35216.041,E2 35216.041} C_VEL
LIN {X 0,Y 744.529,Z 1159.651,A -85,B 0,C 180,E1 35214.264,E2 35214.264} C_VEL
LIN {X 0,Y 744.425,Z 1175.826,A -85,B 0,C 180,E1 35212.757,E2 35212.757} C_VEL
LIN {X 0,Y 744.299,Z 1191.954,A -85,B 0,C 180,E1 35211.102,E2 35211.102} C_VEL
LIN {X 0,Y 744.167,Z 1208.864,A -85,B 0,C 180,E1 35209.138,E2 35209.138} C_VEL
LIN {X 0,Y 744.064,Z 1220.667,A -85,B 0,C 180,E1 35207.599,E2 35207.599} C_VEL
LIN {X 0,Y 744.014,Z 1231.213,A -85,B 0,C 180,E1 35206.072,E2 35206.072} C_VEL
LIN {X 0,Y 744.005,Z 1241.057,A -85,B 0,C 180,E1 35204.476,E2 35204.476} C_VEL
LIN {X 0,Y 743.971,Z 1250.523,A -85,B 0,C 180,E1 35202.733,E2 35202.733} C_VEL
LIN {X 0,Y 743.926,Z 1260.595,A -85,B 0,C 180,E1 35200.532,E2 35200.532} C_VEL
LIN {X 0,Y 743.907,Z 1267.279,A -85,B 0,C 180,E1 35198.736,E2 35198.736} C_VEL
LIN {X 0,Y 743.911,Z 1272.979,A -85,B 0,C 180,E1 35196.87,E2 35196.87} C_VEL
LIN {X 0,Y 743.909,Z 1277.634,A -85,B 0,C 180,E1 35194.78,E2 35194.78} C_VEL
LIN {X 0,Y 743.915,Z 1280.406,A -85,B 0,C 180,E1 35192.851,E2 35192.851} C_VEL
LIN {X 0,Y 743.873,Z 1281.715,A -85,B 0,C 180,E1 35191.001,E2 35191.001} C_VEL
LIN {X 0,Y 743.863,Z 1281.827,A -85,B 0,C 180,E1 35189.384,E2 35189.384} C_VEL
LIN {X 0,Y 743.909,Z 1280.946,A -85,B 0,C 180,E1 35187.766,E2 35187.766} C_VEL
LIN {X 0,Y 743.917,Z 1278.803,A -85,B 0,C 180,E1 35185.915,E2 35185.915} C_VEL
LIN {X 0,Y 743.919,Z 1274.734,A -85,B 0,C 180,E1 35183.827,E2 35183.827} C_VEL
LIN {X 0,Y 743.911,Z 1269.328,A -85,B 0,C 180,E1 35181.887,E2 35181.887} C_VEL
LIN {X 0,Y 743.927,Z 1263.043,A -85,B 0,C 180,E1 35180.094,E2 35180.094} C_VEL
LIN {X 0,Y 743.939,Z 1256.142,A -85,B 0,C 180,E1 35178.448,E2 35178.448} C_VEL
LIN {X 0,Y 743.938,Z 1248.47,A -85,B 0,C 180,E1 35176.871,E2 35176.871} C_VEL
LIN {X 0,Y 743.996,Z 1239.661,A -85,B 0,C 180,E1 35175.286,E2 35175.286} C_VEL
LIN {X 0,Y 744.041,Z 1228.6,A -85,B 0,C 180,E1 35173.528,E2 35173.528} C_VEL
LIN {X 0,Y 744.145,Z 1214.022,A -85,B 0,C 180,E1 35171.512,E2 35171.512} C_VEL
LIN {X 0,Y 744.205,Z 1200.669,A -85,B 0,C 180,E1 35169.882,E2 35169.882} C_VEL
LIN {X 0,Y 744.328,Z 1186.986,A -85,B 0,C 180,E1 35168.373,E2 35168.373} C_VEL
LIN {X 0,Y 744.481,Z 1169.85,A -85,B 0,C 180,E1 35166.659,E2 35166.659} C_VEL
LIN {X 0,Y 744.654,Z 1150.816,A -85,B 0,C 180,E1 35164.978,E2 35164.978} C_VEL
LIN {X 0,Y 744.781,Z 1133.837,A -85,B 0,C 180,E1 35163.617,E2 35163.617} C_VEL
LIN {X 0,Y 745.053,Z 1112.509,A -85,B 0,C 180,E1 35162.072,E2 35162.072} C_VEL
LIN {X 0,Y 745.263,Z 1090.699,A -85,B 0,C 180,E1 35160.679,E2 35160.679} C_VEL
LIN {X 0,Y 745.441,Z 1071.936,A -85,B 0,C 180,E1 35159.597,E2 35159.597} C_VEL
LIN {X 0,Y 745.662,Z 1050.176,A -85,B 0,C 180,E1 35158.469,E2 35158.469} C_VEL
LIN {X 0,Y 745.968,Z 1024.297,A -85,B 0,C 180,E1 35157.305,E2 35157.305} C_VEL
LIN {X 0,Y 746.161,Z 1002.604,A -85,B 0,C 180,E1 35156.461,E2 35156.461} C_VEL
LIN {X 0,Y 746.328,Z 982.56,A -85,B 0,C 180,E1 35155.782,E2 35155.782} C_VEL
LIN {X 0,Y 746.511,Z 960.019,A -85,B 0,C 180,E1 35155.121,E2 35155.121} C_VEL
LIN {X 0,Y 746.689,Z 933.014,A -85,B 0,C 180,E1 35154.49,E2 35154.49} C_VEL
LIN {X 0,Y 746.829,Z 905.664,A -85,B 0,C 180,E1 35154.018,E2 35154.018} C_VEL
LIN {X 0,Y 747.327,Z 662.025,A -85,B 0,C 180,E1 35151.135,E2 35151.135} C_VEL
LIN {X 0,Y 747.723,Z 459.587,A -85,B 0,C 180,E1 35148.669,E2 35148.669} C_VEL
LIN {X 0,Y 747.61,Z 430.206,A -85,B 0,C 180,E1 35148.293,E2 35148.293} C_VEL
LIN {X 0,Y 746.876,Z 426.762,A -85,B 0,C 180,E1 35148.188,E2 35148.188} C_VEL
LIN {X 0,Y 747.196,Z 381.055,A -85,B 0,C 180,E1 35145.53,E2 35145.53} C_VEL
LIN {X 0,Y 747.559,Z 339.555,A -85,B 0,C 180,E1 35143.012,E2 35143.012} C_VEL
LIN {X 0,Y 747.518,Z 336.328,A -85,B 0,C 180,E1 35142.805,E2 35142.805} C_VEL
LIN {X 0,Y 745.704,Z 332.509,A -85,B 0,C 180,E1 35142.412,E2 35142.412} C_VEL
LIN {X 0,Y 744.081,Z 328.958,A -85,B 0,C 180,E1 35142.033,E2 35142.033} C_VEL
LIN {X 0,Y 744.016,Z 328.511,A -85,B 0,C 180,E1 35141.701,E2 35141.701} C_VEL
LIN {X 0,Y 744.01,Z 328.546,A -85,B 0,C 180,E1 35138.911,E2 35138.911} C_VEL
LIN {X 0,Y 744.029,Z 328.537,A -85,B 0,C 180,E1 35136.06,E2 35136.06} C_VEL
LIN {X 0,Y 744.029,Z 328.555,A -85,B 0,C 180,E1 35133.067,E2 35133.067} C_VEL
LIN {X 0,Y 744.035,Z 328.543,A -85,B 0,C 180,E1 35130.067,E2 35130.067} C_VEL
LIN {X 0,Y 744.036,Z 328.554,A -85,B 0,C 180,E1 35127.004,E2 35127.004} C_VEL
LIN {X 0,Y 744.017,Z 328.543,A -85,B 0,C 180,E1 35124.029,E2 35124.029} C_VEL
LIN {X 0,Y 744.024,Z 328.552,A -85,B 0,C 180,E1 35121.11,E2 35121.11} C_VEL
LIN {X 0,Y 744.003,Z 328.549,A -85,B 0,C 180,E1 35118.33,E2 35118.33} C_VEL
LIN {X 0,Y 744.038,Z 328.541,A -85,B 0,C 180,E1 35115.511,E2 35115.511} C_VEL
LIN {X 0,Y 744.025,Z 328.553,A -85,B 0,C 180,E1 35112.496,E2 35112.496} C_VEL
LIN {X 0,Y 744.011,Z 328.544,A -85,B 0,C 180,E1 35109.593,E2 35109.593} C_VEL
LIN {X 0,Y 744.029,Z 328.552,A -85,B 0,C 180,E1 35106.637,E2 35106.637} C_VEL
LIN {X 0,Y 743.996,Z 328.55,A -85,B 0,C 180,E1 35103.853,E2 35103.853} C_VEL
LIN {X 0,Y 744.037,Z 328.541,A -85,B 0,C 180,E1 35101.001,E2 35101.001} C_VEL
LIN {X 0,Y 744.013,Z 328.553,A -85,B 0,C 180,E1 35097.998,E2 35097.998} C_VEL
LIN {X 0,Y 744,Z 328.545,A -85,B 0,C 180,E1 35095.22,E2 35095.22} C_VEL
LIN {X 0,Y 744.029,Z 328.549,A -85,B 0,C 180,E1 35092.354,E2 35092.354} C_VEL
LIN {X 0,Y 744.007,Z 328.553,A -85,B 0,C 180,E1 35091.787,E2 35091.787} C_VEL
LIN {X 0,Y 742.98,Z 328.675,A -85,B 0,C 180,E1 35091.193,E2 35091.193} C_VEL
LIN {X 0,Y 736.566,Z 329.478,A -85,B 0,C 180,E1 35089.532,E2 35089.532} C_VEL
LIN {X 0,Y 736.054,Z 329.536,A -85,B 0,C 180,E1 35089.1,E2 35089.1} C_VEL
LIN {X 0,Y 736.092,Z 329.538,A -85,B 0,C 180,E1 35086.222,E2 35086.222} C_VEL
LIN {X 0,Y 736.056,Z 329.539,A -85,B 0,C 180,E1 35083.425,E2 35083.425} C_VEL
LIN {X 0,Y 736.066,Z 329.534,A -85,B 0,C 180,E1 35080.643,E2 35080.643} C_VEL
LIN {X 0,Y 736.098,Z 329.543,A -85,B 0,C 180,E1 35077.645,E2 35077.645} C_VEL
LIN {X 0,Y 736.042,Z 329.538,A -85,B 0,C 180,E1 35074.836,E2 35074.836} C_VEL
LIN {X 0,Y 736.098,Z 329.533,A -85,B 0,C 180,E1 35072.054,E2 35072.054} C_VEL
LIN {X 0,Y 736.059,Z 329.542,A -85,B 0,C 180,E1 35069.103,E2 35069.103} C_VEL
LIN {X 0,Y 736.042,Z 329.537,A -85,B 0,C 180,E1 35066.434,E2 35066.434} C_VEL
LIN {X 0,Y 736.097,Z 329.536,A -85,B 0,C 180,E1 35063.586,E2 35063.586} C_VEL
LIN {X 0,Y 736.044,Z 329.541,A -85,B 0,C 180,E1 35060.725,E2 35060.725} C_VEL
LIN {X 0,Y 736.041,Z 329.536,A -85,B 0,C 180,E1 35058.11,E2 35058.11} C_VEL
LIN {X 0,Y 736.099,Z 329.542,A -85,B 0,C 180,E1 35055.171,E2 35055.171} C_VEL
LIN {X 0,Y 736.033,Z 329.54,A -85,B 0,C 180,E1 35052.352,E2 35052.352} C_VEL
LIN {X 0,Y 736.043,Z 329.538,A -85,B 0,C 180,E1 35049.779,E2 35049.779} C_VEL
LIN {X 0,Y 736.099,Z 329.543,A -85,B 0,C 180,E1 35046.862,E2 35046.862} C_VEL
LIN {X 0,Y 736.03,Z 329.541,A -85,B 0,C 180,E1 35044.128,E2 35044.128} C_VEL
LIN {X 0,Y 736.033,Z 329.538,A -85,B 0,C 180,E1 35041.595,E2 35041.595} C_VEL
LIN {X 0,Y 736.1,Z 329.539,A -85,B 0,C 180,E1 35038.741,E2 35038.741} C_VEL
LIN {X 0,Y 736.029,Z 329.541,A -85,B 0,C 180,E1 35035.93,E2 35035.93} C_VEL
LIN {X 0,Y 736.022,Z 329.538,A -85,B 0,C 180,E1 35033.455,E2 35033.455} C_VEL
LIN {X 0,Y 736.098,Z 329.537,A -85,B 0,C 180,E1 35030.681,E2 35030.681} C_VEL
LIN {X 0,Y 736.029,Z 329.542,A -85,B 0,C 180,E1 35027.766,E2 35027.766} C_VEL
LIN {X 0,Y 736.015,Z 329.54,A -85,B 0,C 180,E1 35025.301,E2 35025.301} C_VEL
LIN {X 0,Y 736.048,Z 329.539,A -85,B 0,C 180,E1 35022.741,E2 35022.741} C_VEL
LIN {X 0,Y 736.041,Z 329.544,A -85,B 0,C 180,E1 35019.698,E2 35019.698} C_VEL
LIN {X 0,Y 736.011,Z 329.542,A -85,B 0,C 180,E1 35017.258,E2 35017.258} C_VEL
LIN {X 0,Y 736.01,Z 329.54,A -85,B 0,C 180,E1 35014.91,E2 35014.91} C_VEL
LIN {X 0,Y 736.067,Z 329.539,A -85,B 0,C 180,E1 35012.258,E2 35012.258} C_VEL
LIN {X 0,Y 736.026,Z 329.544,A -85,B 0,C 180,E1 35009.299,E2 35009.299} C_VEL
LIN {X 0,Y 736.003,Z 329.539,A -85,B 0,C 180,E1 35006.885,E2 35006.885} C_VEL
LIN {X 0,Y 736.003,Z 329.543,A -85,B 0,C 180,E1 35004.621,E2 35004.621} C_VEL
LIN {X 0,Y 736.035,Z 329.539,A -85,B 0,C 180,E1 35002.114,E2 35002.114} C_VEL
LIN {X 0,Y 736.024,Z 329.543,A -85,B 0,C 180,E1 34999.036,E2 34999.036} C_VEL
LIN {X 0,Y 735.997,Z 329.542,A -85,B 0,C 180,E1 34996.588,E2 34996.588} C_VEL
LIN {X 0,Y 735.994,Z 329.526,A -85,B 0,C 180,E1 34994.315,E2 34994.315} C_VEL
LIN {X 0,Y 736.01,Z 329.546,A -85,B 0,C 180,E1 34991.956,E2 34991.956} C_VEL
LIN {X 0,Y 736.053,Z 329.54,A -85,B 0,C 180,E1 34988.984,E2 34988.984} C_VEL
LIN {X 0,Y 736.076,Z 329.704,A -85,B 0,C 180,E1 34986.931,E2 34986.931} C_VEL
LIN {X 0,Y 736.413,Z 331.162,A -85,B 0,C 180,E1 34986.791,E2 34986.791} C_VEL
LIN {X 0,Y 738.265,Z 334.163,A -85,B 0,C 180,E1 34986.62,E2 34986.62} C_VEL
LIN {X 0,Y 739.581,Z 336.012,A -85,B 0,C 180,E1 34986.506,E2 34986.506} C_VEL
LIN {X 0,Y 741.645,Z 339.464,A -85,B 0,C 180,E1 34986.321,E2 34986.321} C_VEL
LIN {X 0,Y 740.955,Z 555.844,A -85,B 0,C 180,E1 34983.683,E2 34983.683} C_VEL
LIN {X 0,Y 740.33,Z 756.433,A -85,B 0,C 180,E1 34981.292,E2 34981.292} C_VEL
LIN {X 0,Y 740.131,Z 783.13,A -85,B 0,C 180,E1 34980.825,E2 34980.825} C_VEL
LIN {X 0,Y 739.858,Z 810.315,A -85,B 0,C 180,E1 34980.186,E2 34980.186} C_VEL
LIN {X 0,Y 739.579,Z 833.792,A -85,B 0,C 180,E1 34979.492,E2 34979.492} C_VEL
LIN {X 0,Y 739.289,Z 857.588,A -85,B 0,C 180,E1 34978.666,E2 34978.666} C_VEL
LIN {X 0,Y 738.843,Z 883.632,A -85,B 0,C 180,E1 34977.595,E2 34977.595} C_VEL
LIN {X 0,Y 738.514,Z 905.378,A -85,B 0,C 180,E1 34976.562,E2 34976.562} C_VEL
LIN {X 0,Y 738.213,Z 926.679,A -85,B 0,C 180,E1 34975.423,E2 34975.423} C_VEL
LIN {X 0,Y 737.784,Z 951.485,A -85,B 0,C 180,E1 34973.92,E2 34973.92} C_VEL
LIN {X 0,Y 737.466,Z 970.827,A -85,B 0,C 180,E1 34972.598,E2 34972.598} C_VEL
LIN {X 0,Y 737.214,Z 991.261,A -85,B 0,C 180,E1 34971.05,E2 34971.05} C_VEL
LIN {X 0,Y 736.858,Z 1011.316,A -85,B 0,C 180,E1 34969.336,E2 34969.336} C_VEL
LIN {X 0,Y 736.678,Z 1027.257,A -85,B 0,C 180,E1 34967.824,E2 34967.824} C_VEL
LIN {X 0,Y 736.458,Z 1044.963,A -85,B 0,C 180,E1 34965.962,E2 34965.962} C_VEL
LIN {X 0,Y 736.283,Z 1060.007,A -85,B 0,C 180,E1 34964.161,E2 34964.161} C_VEL
LIN {X 0,Y 736.191,Z 1072,A -85,B 0,C 180,E1 34962.562,E2 34962.562} C_VEL
LIN {X 0,Y 736.07,Z 1083.178,A -85,B 0,C 180,E1 34960.902,E2 34960.902} C_VEL
LIN {X 0,Y 736.025,Z 1095.154,A -85,B 0,C 180,E1 34958.876,E2 34958.876} C_VEL
LIN {X 0,Y 735.925,Z 1104.915,A -85,B 0,C 180,E1 34956.909,E2 34956.909} C_VEL
LIN {X 0,Y 735.918,Z 1111.939,A -85,B 0,C 180,E1 34955.258,E2 34955.258} C_VEL
LIN {X 0,Y 735.931,Z 1117.985,A -85,B 0,C 180,E1 34953.572,E2 34953.572} C_VEL
LIN {X 0,Y 735.912,Z 1123.42,A -85,B 0,C 180,E1 34951.724,E2 34951.724} C_VEL
LIN {X 0,Y 735.907,Z 1127.905,A -85,B 0,C 180,E1 34949.642,E2 34949.642} C_VEL
LIN {X 0,Y 735.896,Z 1130.584,A -85,B 0,C 180,E1 34947.64,E2 34947.64} C_VEL
LIN {X 0,Y 735.913,Z 1131.752,A -85,B 0,C 180,E1 34945.858,E2 34945.858} C_VEL
LIN {X 0,Y 735.887,Z 1131.778,A -85,B 0,C 180,E1 34944.141,E2 34944.141} C_VEL
LIN {X 0,Y 735.878,Z 1130.737,A -85,B 0,C 180,E1 34942.446,E2 34942.446} C_VEL
LIN {X 0,Y 735.913,Z 1128.42,A -85,B 0,C 180,E1 34940.588,E2 34940.588} C_VEL
LIN {X 0,Y 735.919,Z 1124.297,A -85,B 0,C 180,E1 34938.538,E2 34938.538} C_VEL
LIN {X 0,Y 735.911,Z 1118.769,A -85,B 0,C 180,E1 34936.579,E2 34936.579} C_VEL
LIN {X 0,Y 735.937,Z 1112.817,A -85,B 0,C 180,E1 34934.88,E2 34934.88} C_VEL
LIN {X 0,Y 735.951,Z 1105.78,A -85,B 0,C 180,E1 34933.194,E2 34933.194} C_VEL
LIN {X 0,Y 735.999,Z 1097.647,A -85,B 0,C 180,E1 34931.52,E2 34931.52} C_VEL
LIN {X 0,Y 736.065,Z 1087.014,A -85,B 0,C 180,E1 34929.619,E2 34929.619} C_VEL
LIN {X 0,Y 736.163,Z 1073.598,A -85,B 0,C 180,E1 34927.571,E2 34927.571} C_VEL
LIN {X 0,Y 736.264,Z 1061.383,A -85,B 0,C 180,E1 34925.924,E2 34925.924} C_VEL
LIN {X 0,Y 736.414,Z 1048.5,A -85,B 0,C 180,E1 34924.361,E2 34924.361} C_VEL
LIN {X 0,Y 736.647,Z 1031.346,A -85,B 0,C 180,E1 34922.489,E2 34922.489} C_VEL
LIN {X 0,Y 736.861,Z 1013.551,A -85,B 0,C 180,E1 34920.778,E2 34920.778} C_VEL
LIN {X 0,Y 737.106,Z 995.69,A -85,B 0,C 180,E1 34919.223,E2 34919.223} C_VEL
LIN {X 0,Y 737.437,Z 973.604,A -85,B 0,C 180,E1 34917.513,E2 34917.513} C_VEL
LIN {X 0,Y 737.73,Z 954.539,A -85,B 0,C 180,E1 34916.192,E2 34916.192} C_VEL
LIN {X 0,Y 738.13,Z 932.08,A -85,B 0,C 180,E1 34914.793,E2 34914.793} C_VEL
LIN {X 0,Y 738.489,Z 907.749,A -85,B 0,C 180,E1 34913.469,E2 34913.469} C_VEL
LIN {X 0,Y 738.797,Z 887.58,A -85,B 0,C 180,E1 34912.496,E2 34912.496} C_VEL
LIN {X 0,Y 739.126,Z 864.727,A -85,B 0,C 180,E1 34911.52,E2 34911.52} C_VEL
LIN {X 0,Y 739.543,Z 837.771,A -85,B 0,C 180,E1 34910.545,E2 34910.545} C_VEL
LIN {X 0,Y 739.836,Z 812.305,A -85,B 0,C 180,E1 34909.778,E2 34909.778} C_VEL
LIN {X 0,Y 740.098,Z 785.271,A -85,B 0,C 180,E1 34909.13,E2 34909.13} C_VEL
LIN {X 0,Y 740.319,Z 759.135,A -85,B 0,C 180,E1 34908.658,E2 34908.658} C_VEL
LIN {X 0,Y 740.502,Z 711.721,A -85,B 0,C 180,E1 34908.073,E2 34908.073} C_VEL
LIN {X 0,Y 741.177,Z 485.861,A -85,B 0,C 180,E1 34905.384,E2 34905.384} C_VEL
LIN {X 0,Y 741.565,Z 338.952,A -85,B 0,C 180,E1 34903.577,E2 34903.577} C_VEL
LIN {X 0,Y 738.56,Z 334.427,A -85,B 0,C 180,E1 34903.314,E2 34903.314} C_VEL
LIN {X 0,Y 736.517,Z 331.4,A -85,B 0,C 180,E1 34903.131,E2 34903.131} C_VEL
LIN {X 0,Y 736.103,Z 329.799,A -85,B 0,C 180,E1 34902.993,E2 34902.993} C_VEL
LIN {X 0,Y 736.026,Z 329.547,A -85,B 0,C 180,E1 34901.629,E2 34901.629} C_VEL
LIN {X 0,Y 736.063,Z 329.53,A -85,B 0,C 180,E1 34898.984,E2 34898.984} C_VEL
LIN {X 0,Y 736.062,Z 329.538,A -85,B 0,C 180,E1 34895.902,E2 34895.902} C_VEL
LIN {X 0,Y 736.049,Z 329.542,A -85,B 0,C 180,E1 34893.188,E2 34893.188} C_VEL
LIN {X 0,Y 736.092,Z 329.54,A -85,B 0,C 180,E1 34890.366,E2 34890.366} C_VEL
LIN {X 0,Y 736.063,Z 329.537,A -85,B 0,C 180,E1 34887.519,E2 34887.519} C_VEL
LIN {X 0,Y 736.097,Z 329.544,A -85,B 0,C 180,E1 34884.643,E2 34884.643} C_VEL
LIN {X 0,Y 736.089,Z 329.537,A -85,B 0,C 180,E1 34881.607,E2 34881.607} C_VEL
LIN {X 0,Y 736.106,Z 329.643,A -85,B 0,C 180,E1 34878.656,E2 34878.656} C_VEL
LIN {X 0,Y 736.756,Z 331.85,A -85,B 0,C 180,E1 34878.398,E2 34878.398} C_VEL
LIN {X 0,Y 738.689,Z 335.428,A -85,B 0,C 180,E1 34877.997,E2 34877.997} C_VEL
LIN {X 0,Y 741.435,Z 341.007,A -85,B 0,C 180,E1 34877.405,E2 34877.405} C_VEL
LIN {X 0,Y 740.891,Z 382.846,A -85,B 0,C 180,E1 34874.841,E2 34874.841} C_VEL
LIN {X 0,Y 740.508,Z 427.348,A -85,B 0,C 180,E1 34872.239,E2 34872.239} C_VEL
LIN {X 0,Y 741.786,Z 433.879,A -85,B 0,C 180,E1 34872.063,E2 34872.063} C_VEL
LIN {X 0,Y 741.149,Z 644.067,A -85,B 0,C 180,E1 34869.472,E2 34869.472} C_VEL
LIN {X 0,Y 740.484,Z 870.072,A -85,B 0,C 180,E1 34866.783,E2 34866.783} C_VEL
LIN {X 0,Y 740.319,Z 910.027,A -85,B 0,C 180,E1 34866.283,E2 34866.283} C_VEL
LIN {X 0,Y 740.076,Z 936.604,A -85,B 0,C 180,E1 34865.797,E2 34865.797} C_VEL
LIN {X 0,Y 739.821,Z 962.716,A -85,B 0,C 180,E1 34865.166,E2 34865.166} C_VEL
LIN {X 0,Y 739.525,Z 989.895,A -85,B 0,C 180,E1 34864.343,E2 34864.343} C_VEL
LIN {X 0,Y 739.109,Z 1015.356,A -85,B 0,C 180,E1 34863.408,E2 34863.408} C_VEL
LIN {X 0,Y 738.798,Z 1036.689,A -85,B 0,C 180,E1 34862.499,E2 34862.499} C_VEL
LIN {X 0,Y 738.502,Z 1056.411,A -85,B 0,C 180,E1 34861.553,E2 34861.553} C_VEL
LIN {X 0,Y 738.186,Z 1078.846,A -85,B 0,C 180,E1 34860.347,E2 34860.347} C_VEL
LIN {X 0,Y 737.755,Z 1102.589,A -85,B 0,C 180,E1 34858.891,E2 34858.891} C_VEL
LIN {X 0,Y 737.473,Z 1121.044,A -85,B 0,C 180,E1 34857.625,E2 34857.625} C_VEL
LIN {X 0,Y 737.206,Z 1139.928,A -85,B 0,C 180,E1 34856.198,E2 34856.198} C_VEL
LIN {X 0,Y 736.866,Z 1160.583,A -85,B 0,C 180,E1 34854.448,E2 34854.448} C_VEL
LIN {X 0,Y 736.694,Z 1175.828,A -85,B 0,C 180,E1 34853.01,E2 34853.01} C_VEL
LIN {X 0,Y 736.505,Z 1191.956,A -85,B 0,C 180,E1 34851.336,E2 34851.336} C_VEL
LIN {X 0,Y 736.308,Z 1208.866,A -85,B 0,C 180,E1 34849.35,E2 34849.35} C_VEL
LIN {X 0,Y 736.17,Z 1220.669,A -85,B 0,C 180,E1 34847.794,E2 34847.794} C_VEL
LIN {X 0,Y 736.087,Z 1231.215,A -85,B 0,C 180,E1 34846.25,E2 34846.25} C_VEL
LIN {X 0,Y 736.048,Z 1241.059,A -85,B 0,C 180,E1 34844.635,E2 34844.635} C_VEL
LIN {X 0,Y 735.992,Z 1250.524,A -85,B 0,C 180,E1 34842.874,E2 34842.874} C_VEL
LIN {X 0,Y 735.933,Z 1260.596,A -85,B 0,C 180,E1 34840.648,E2 34840.648} C_VEL
LIN {X 0,Y 735.903,Z 1267.28,A -85,B 0,C 180,E1 34838.832,E2 34838.832} C_VEL
LIN {X 0,Y 735.915,Z 1272.979,A -85,B 0,C 180,E1 34836.945,E2 34836.945} C_VEL
LIN {X 0,Y 735.911,Z 1277.634,A -85,B 0,C 180,E1 34834.832,E2 34834.832} C_VEL
LIN {X 0,Y 735.914,Z 1280.406,A -85,B 0,C 180,E1 34832.882,E2 34832.882} C_VEL
LIN {X 0,Y 735.873,Z 1281.715,A -85,B 0,C 180,E1 34831.012,E2 34831.012} C_VEL
LIN {X 0,Y 735.863,Z 1281.827,A -85,B 0,C 180,E1 34829.377,E2 34829.377} C_VEL
LIN {X 0,Y 735.907,Z 1280.946,A -85,B 0,C 180,E1 34827.742,E2 34827.742} C_VEL
LIN {X 0,Y 735.918,Z 1278.803,A -85,B 0,C 180,E1 34825.871,E2 34825.871} C_VEL
LIN {X 0,Y 735.922,Z 1274.734,A -85,B 0,C 180,E1 34823.76,E2 34823.76} C_VEL
LIN {X 0,Y 735.934,Z 1269.072,A -85,B 0,C 180,E1 34821.72,E2 34821.72} C_VEL
LIN {X 0,Y 735.945,Z 1263.044,A -85,B 0,C 180,E1 34819.985,E2 34819.985} C_VEL
LIN {X 0,Y 735.951,Z 1256.144,A -85,B 0,C 180,E1 34818.321,E2 34818.321} C_VEL
LIN {X 0,Y 735.966,Z 1248.882,A -85,B 0,C 180,E1 34816.806,E2 34816.806} C_VEL
LIN {X 0,Y 736.041,Z 1240.128,A -85,B 0,C 180,E1 34815.203,E2 34815.203} C_VEL
LIN {X 0,Y 736.106,Z 1229.835,A -85,B 0,C 180,E1 34813.537,E2 34813.537} C_VEL
LIN {X 0,Y 736.26,Z 1215.947,A -85,B 0,C 180,E1 34811.553,E2 34811.553} C_VEL
LIN {X 0,Y 736.374,Z 1201.381,A -85,B 0,C 180,E1 34809.742,E2 34809.742} C_VEL
LIN {X 0,Y 736.537,Z 1187.744,A -85,B 0,C 180,E1 34808.213,E2 34808.213} C_VEL
LIN {X 0,Y 736.752,Z 1171.419,A -85,B 0,C 180,E1 34806.555,E2 34806.555} C_VEL
LIN {X 0,Y 737.035,Z 1151.831,A -85,B 0,C 180,E1 34804.787,E2 34804.787} C_VEL
LIN {X 0,Y 737.239,Z 1134.945,A -85,B 0,C 180,E1 34803.413,E2 34803.413} C_VEL
LIN {X 0,Y 737.583,Z 1115.598,A -85,B 0,C 180,E1 34801.984,E2 34801.984} C_VEL
LIN {X 0,Y 737.954,Z 1092.087,A -85,B 0,C 180,E1 34800.445,E2 34800.445} C_VEL
LIN {X 0,Y 738.233,Z 1072.421,A -85,B 0,C 180,E1 34799.295,E2 34799.295} C_VEL
LIN {X 0,Y 738.553,Z 1051.959,A -85,B 0,C 180,E1 34798.221,E2 34798.221} C_VEL
LIN {X 0,Y 739.02,Z 1025.792,A -85,B 0,C 180,E1 34797.02,E2 34797.02} C_VEL
LIN {X 0,Y 739.316,Z 1003.386,A -85,B 0,C 180,E1 34796.137,E2 34796.137} C_VEL
LIN {X 0,Y 739.58,Z 982.461,A -85,B 0,C 180,E1 34795.422,E2 34795.422} C_VEL
LIN {X 0,Y 739.855,Z 959.894,A -85,B 0,C 180,E1 34794.758,E2 34794.758} C_VEL
LIN {X 0,Y 740.128,Z 933.025,A -85,B 0,C 180,E1 34794.128,E2 34794.128} C_VEL
LIN {X 0,Y 740.333,Z 905.664,A -85,B 0,C 180,E1 34793.652,E2 34793.652} C_VEL
LIN {X 0,Y 741.077,Z 664.836,A -85,B 0,C 180,E1 34790.779,E2 34790.779} C_VEL
LIN {X 0,Y 741.694,Z 462.514,A -85,B 0,C 180,E1 34788.296,E2 34788.296} C_VEL
LIN {X 0,Y 741.609,Z 432.191,A -85,B 0,C 180,E1 34787.903,E2 34787.903} C_VEL
LIN {X 0,Y 740.423,Z 426.676,A -85,B 0,C 180,E1 34787.735,E2 34787.735} C_VEL
LIN {X 0,Y 740.903,Z 381.95,A -85,B 0,C 180,E1 34785.105,E2 34785.105} C_VEL
LIN {X 0,Y 741.435,Z 341.007,A -85,B 0,C 180,E1 34782.595,E2 34782.595} C_VEL
LIN {X 0,Y 739.569,Z 337.216,A -85,B 0,C 180,E1 34782.194,E2 34782.194} C_VEL
LIN {X 0,Y 737.862,Z 333.633,A -85,B 0,C 180,E1 34781.815,E2 34781.815} C_VEL
LIN {X 0,Y 736.185,Z 330.067,A -85,B 0,C 180,E1 34781.424,E2 34781.424} C_VEL
LIN {X 0,Y 736.077,Z 329.499,A -85,B 0,C 180,E1 34781.189,E2 34781.189} C_VEL
LIN {X 0,Y 736.094,Z 329.519,A -85,B 0,C 180,E1 34778.268,E2 34778.268} C_VEL
LIN {X 0,Y 736.091,Z 329.54,A -85,B 0,C 180,E1 34775.167,E2 34775.167} C_VEL
LIN {X 0,Y 736.089,Z 329.534,A -85,B 0,C 180,E1 34772.174,E2 34772.174} C_VEL
LIN {X 0,Y 736.098,Z 329.542,A -85,B 0,C 180,E1 34769.097,E2 34769.097} C_VEL
LIN {X 0,Y 736.078,Z 329.533,A -85,B 0,C 180,E1 34766.112,E2 34766.112} C_VEL
LIN {X 0,Y 736.085,Z 329.539,A -85,B 0,C 180,E1 34763.2,E2 34763.2} C_VEL
LIN {X 0,Y 736.064,Z 329.539,A -85,B 0,C 180,E1 34760.35,E2 34760.35} C_VEL
LIN {X 0,Y 736.097,Z 329.53,A -85,B 0,C 180,E1 34757.53,E2 34757.53} C_VEL
LIN {X 0,Y 736.08,Z 329.543,A -85,B 0,C 180,E1 34754.474,E2 34754.474} C_VEL
LIN {X 0,Y 736.085,Z 329.531,A -85,B 0,C 180,E1 34751.518,E2 34751.518} C_VEL
LIN {X 0,Y 736.091,Z 329.543,A -85,B 0,C 180,E1 34748.436,E2 34748.436} C_VEL
LIN {X 0,Y 736.065,Z 329.533,A -85,B 0,C 180,E1 34745.535,E2 34745.535} C_VEL
LIN {X 0,Y 736.088,Z 329.539,A -85,B 0,C 180,E1 34742.647,E2 34742.647} C_VEL
LIN {X 0,Y 736.06,Z 329.54,A -85,B 0,C 180,E1 34739.844,E2 34739.844} C_VEL
LIN {X 0,Y 736.083,Z 329.532,A -85,B 0,C 180,E1 34737.041,E2 34737.041} C_VEL
LIN {X 0,Y 736.078,Z 329.542,A -85,B 0,C 180,E1 34733.918,E2 34733.918} C_VEL
LIN {X 0,Y 736.059,Z 329.535,A -85,B 0,C 180,E1 34731.091,E2 34731.091} C_VEL
LIN {X 0,Y 736.054,Z 329.536,A -85,B 0,C 180,E1 34729.1,E2 34729.1} C_VEL
LIN {X 0,Y 735.095,Z 329.659,A -85,B 0,C 180,E1 34728.5,E2 34728.5} C_VEL
LIN {X 0,Y 728.699,Z 330.454,A -85,B 0,C 180,E1 34726.821,E2 34726.821} C_VEL
LIN {X 0,Y 728.156,Z 330.524,A -85,B 0,C 180,E1 34726.385,E2 34726.385} C_VEL
LIN {X 0,Y 728.119,Z 330.528,A -85,B 0,C 180,E1 34723.438,E2 34723.438} C_VEL
LIN {X 0,Y 728.128,Z 330.523,A -85,B 0,C 180,E1 34720.63,E2 34720.63} C_VEL
LIN {X 0,Y 728.145,Z 330.531,A -85,B 0,C 180,E1 34717.541,E2 34717.541} C_VEL
LIN {X 0,Y 728.104,Z 330.527,A -85,B 0,C 180,E1 34714.804,E2 34714.804} C_VEL
LIN {X 0,Y 728.162,Z 330.523,A -85,B 0,C 180,E1 34711.99,E2 34711.99} C_VEL
LIN {X 0,Y 728.12,Z 330.531,A -85,B 0,C 180,E1 34709.096,E2 34709.096} C_VEL
LIN {X 0,Y 728.105,Z 330.526,A -85,B 0,C 180,E1 34706.397,E2 34706.397} C_VEL
LIN {X 0,Y 728.158,Z 330.526,A -85,B 0,C 180,E1 34703.517,E2 34703.517} C_VEL
LIN {X 0,Y 728.101,Z 330.529,A -85,B 0,C 180,E1 34700.637,E2 34700.637} C_VEL
LIN {X 0,Y 728.108,Z 330.525,A -85,B 0,C 180,E1 34698.026,E2 34698.026} C_VEL
LIN {X 0,Y 728.154,Z 330.532,A -85,B 0,C 180,E1 34695.006,E2 34695.006} C_VEL
LIN {X 0,Y 728.092,Z 330.528,A -85,B 0,C 180,E1 34692.25,E2 34692.25} C_VEL
LIN {X 0,Y 728.119,Z 330.526,A -85,B 0,C 180,E1 34689.61,E2 34689.61} C_VEL
LIN {X 0,Y 728.115,Z 330.531,A -85,B 0,C 180,E1 34686.485,E2 34686.485} C_VEL
LIN {X 0,Y 728.087,Z 330.529,A -85,B 0,C 180,E1 34683.887,E2 34683.887} C_VEL
LIN {X 0,Y 728.124,Z 330.525,A -85,B 0,C 180,E1 34681.27,E2 34681.27} C_VEL
